LIN {X 0,Y 573.253,Z 369.075,A -85,B 0,C 180,E1 -2323.622,E2 -2323.622} C_VEL
LIN {X 0,Y 573.279,Z 369.074,A -85,B 0,C 180,E1 -2325.807,E2 -2325.807} C_VEL
LIN {X 0,Y 573.268,Z 369.074,A -85,B 0,C 180,E1 -2328.745,E2 -2328.745} C_VEL
LIN {X 0,Y 573.293,Z 369.076,A -85,B 0,C 180,E1 -2331.541,E2 -2331.541} C_VEL
LIN {X 0,Y 573.293,Z 369.073,A -85,B 0,C 180,E1 -2334.372,E2 -2334.372} C_VEL
LIN {X 0,Y 573.313,Z 369.07,A -85,B 0,C 180,E1 -2337.892,E2 -2337.892} C_VEL
LIN {X 0,Y 573.334,Z 369.065,A -85,B 0,C 180,E1 -2340.702,E2 -2340.702} C_VEL
LIN {X 0,Y 573.234,Z 369.083,A -85,B 0,C 180,E1 -2343.515,E2 -2343.515} C_VEL
LIN {X 0,Y 573.294,Z 369.071,A -85,B 0,C 180,E1 -2345.628,E2 -2345.628} C_VEL
LIN {X 0,Y 573.276,Z 369.072,A -85,B 0,C 180,E1 -2347.75,E2 -2347.75} C_VEL
LIN {X 0,Y 573.269,Z 369.075,A -85,B 0,C 180,E1 -2350.597,E2 -2350.597} C_VEL
LIN {X 0,Y 573.268,Z 369.073,A -85,B 0,C 180,E1 -2352.749,E2 -2352.749} C_VEL
LIN {X 0,Y 573.239,Z 369.079,A -85,B 0,C 180,E1 -2354.92,E2 -2354.92} C_VEL
LIN {X 0,Y 573.243,Z 369.077,A -85,B 0,C 180,E1 -2357.849,E2 -2357.849} C_VEL
LIN {X 0,Y 573.258,Z 369.077,A -85,B 0,C 180,E1 -2360.077,E2 -2360.077} C_VEL
LIN {X 0,Y 573.239,Z 369.076,A -85,B 0,C 180,E1 -2363.099,E2 -2363.099} C_VEL
LIN {X 0,Y 573.254,Z 369.076,A -85,B 0,C 180,E1 -2364.389,E2 -2364.389} C_VEL
LIN {X 0,Y 572.629,Z 369.154,A -85,B 0,C 180,E1 -2364.975,E2 -2364.975} C_VEL
LIN {X 0,Y 569.787,Z 369.513,A -85,B 0,C 180,E1 -2365.926,E2 -2365.926} C_VEL
LIN {X 0,Y 567.353,Z 369.819,A -85,B 0,C 180,E1 -2366.692,E2 -2366.692} C_VEL
LIN {X 0,Y 566.297,Z 369.948,A -85,B 0,C 180,E1 -2367.283,E2 -2367.283} C_VEL
LIN {X 0,Y 566.207,Z 369.957,A -85,B 0,C 180,E1 -2367.483,E2 -2367.483} C_VEL
LIN {X 0,Y 566.205,Z 369.954,A -85,B 0,C 180,E1 -2369.769,E2 -2369.769} C_VEL
LIN {X 0,Y 566.208,Z 369.959,A -85,B 0,C 180,E1 -2372.43,E2 -2372.43} C_VEL
LIN {X 0,Y 566.186,Z 369.955,A -85,B 0,C 180,E1 -2374.99,E2 -2374.99} C_VEL
LIN {X 0,Y 566.2,Z 369.959,A -85,B 0,C 180,E1 -2377.461,E2 -2377.461} C_VEL
LIN {X 0,Y 566.222,Z 369.951,A -85,B 0,C 180,E1 -2380.198,E2 -2380.198} C_VEL
LIN {X 0,Y 566.203,Z 369.957,A -85,B 0,C 180,E1 -2383.054,E2 -2383.054} C_VEL
LIN {X 0,Y 566.206,Z 369.96,A -85,B 0,C 180,E1 -2386.048,E2 -2386.048} C_VEL
LIN {X 0,Y 566.186,Z 369.955,A -85,B 0,C 180,E1 -2388.861,E2 -2388.861} C_VEL
LIN {X 0,Y 566.19,Z 369.958,A -85,B 0,C 180,E1 -2391.637,E2 -2391.637} C_VEL
LIN {X 0,Y 566.135,Z 369.965,A -85,B 0,C 180,E1 -2394.306,E2 -2394.306} C_VEL
LIN {X 0,Y 566.112,Z 369.972,A -85,B 0,C 180,E1 -2395.175,E2 -2395.175} C_VEL
LIN {X 0,Y 566.066,Z 370.716,A -85,B 0,C 180,E1 -2396.289,E2 -2396.289} C_VEL
LIN {X 0,Y 566.04,Z 373.544,A -85,B 0,C 180,E1 -2398.95,E2 -2398.95} C_VEL
LIN {X 0,Y 565.999,Z 376.682,A -85,B 0,C 180,E1 -2401.846,E2 -2401.846} C_VEL
LIN {X 0,Y 565.988,Z 379.352,A -85,B 0,C 180,E1 -2404.24,E2 -2404.24} C_VEL
LIN {X 0,Y 565.896,Z 382.829,A -85,B 0,C 180,E1 -2407.356,E2 -2407.356} C_VEL
LIN {X 0,Y 565.884,Z 385.612,A -85,B 0,C 180,E1 -2409.65,E2 -2409.65} C_VEL
LIN {X 0,Y 565.864,Z 389.455,A -85,B 0,C 180,E1 -2412.658,E2 -2412.658} C_VEL
LIN {X 0,Y 565.893,Z 393.314,A -85,B 0,C 180,E1 -2415.63,E2 -2415.63} C_VEL
LIN {X 0,Y 565.897,Z 395.671,A -85,B 0,C 180,E1 -2417.425,E2 -2417.425} C_VEL
LIN {X 0,Y 566.89,Z 403.279,A -85,B 0,C 180,E1 -2417.629,E2 -2417.629} C_VEL
LIN {X 0,Y 566.772,Z 415.78,A -85,B 0,C 180,E1 -2418.013,E2 -2418.013} C_VEL
LIN {X 0,Y 566.661,Z 428.299,A -85,B 0,C 180,E1 -2418.554,E2 -2418.554} C_VEL
LIN {X 0,Y 566.512,Z 439.58,A -85,B 0,C 180,E1 -2419.192,E2 -2419.192} C_VEL
LIN {X 0,Y 566.349,Z 450.842,A -85,B 0,C 180,E1 -2419.995,E2 -2419.995} C_VEL
LIN {X 0,Y 566.238,Z 460.89,A -85,B 0,C 180,E1 -2420.895,E2 -2420.895} C_VEL
LIN {X 0,Y 566.113,Z 470.591,A -85,B 0,C 180,E1 -2421.972,E2 -2421.972} C_VEL
LIN {X 0,Y 566.05,Z 477.159,A -85,B 0,C 180,E1 -2422.868,E2 -2422.868} C_VEL
LIN {X 0,Y 566.003,Z 483.628,A -85,B 0,C 180,E1 -2423.942,E2 -2423.942} C_VEL
LIN {X 0,Y 565.877,Z 488.765,A -85,B 0,C 180,E1 -2425.013,E2 -2425.013} C_VEL
LIN {X 0,Y 565.926,Z 492.754,A -85,B 0,C 180,E1 -2426.084,E2 -2426.084} C_VEL
LIN {X 0,Y 565.877,Z 495.702,A -85,B 0,C 180,E1 -2427.153,E2 -2427.153} C_VEL
LIN {X 0,Y 565.841,Z 497.128,A -85,B 0,C 180,E1 -2427.865,E2 -2427.865} C_VEL
LIN {X 0,Y 565.841,Z 498.756,A -85,B 0,C 180,E1 -2429.288,E2 -2429.288} C_VEL
LIN {X 0,Y 565.839,Z 498.996,A -85,B 0,C 180,E1 -2430,E2 -2430} C_VEL
LIN {X 0,Y 565.841,Z 498.814,A -85,B 0,C 180,E1 -2430.712,E2 -2430.712} C_VEL
LIN {X 0,Y 565.841,Z 497.268,A -85,B 0,C 180,E1 -2432.135,E2 -2432.135} C_VEL
LIN {X 0,Y 565.878,Z 495.907,A -85,B 0,C 180,E1 -2432.848,E2 -2432.848} C_VEL
LIN {X 0,Y 565.926,Z 493.03,A -85,B 0,C 180,E1 -2433.917,E2 -2433.917} C_VEL
LIN {X 0,Y 565.878,Z 489.129,A -85,B 0,C 180,E1 -2434.988,E2 -2434.988} C_VEL
LIN {X 0,Y 565.991,Z 484.096,A -85,B 0,C 180,E1 -2436.059,E2 -2436.059} C_VEL
LIN {X 0,Y 566.031,Z 477.771,A -85,B 0,C 180,E1 -2437.133,E2 -2437.133} C_VEL
LIN {X 0,Y 566.128,Z 469.849,A -85,B 0,C 180,E1 -2438.208,E2 -2438.208} C_VEL
LIN {X 0,Y 566.249,Z 459.997,A -85,B 0,C 180,E1 -2439.285,E2 -2439.285} C_VEL
LIN {X 0,Y 566.426,Z 449.677,A -85,B 0,C 180,E1 -2440.184,E2 -2440.184} C_VEL
LIN {X 0,Y 566.537,Z 438.407,A -85,B 0,C 180,E1 -2440.972,E2 -2440.972} C_VEL
LIN {X 0,Y 566.659,Z 427.185,A -85,B 0,C 180,E1 -2441.593,E2 -2441.593} C_VEL
LIN {X 0,Y 566.781,Z 414.589,A -85,B 0,C 180,E1 -2442.119,E2 -2442.119} C_VEL
LIN {X 0,Y 566.818,Z 401.411,A -85,B 0,C 180,E1 -2442.509,E2 -2442.509} C_VEL
LIN {X 0,Y 565.899,Z 395.669,A -85,B 0,C 180,E1 -2442.667,E2 -2442.667} C_VEL
LIN {X 0,Y 565.855,Z 392.455,A -85,B 0,C 180,E1 -2445.119,E2 -2445.119} C_VEL
LIN {X 0,Y 565.864,Z 389.571,A -85,B 0,C 180,E1 -2447.342,E2 -2447.342} C_VEL
LIN {X 0,Y 565.884,Z 385.726,A -85,B 0,C 180,E1 -2450.35,E2 -2450.35} C_VEL
LIN {X 0,Y 565.91,Z 382.308,A -85,B 0,C 180,E1 -2453.219,E2 -2453.219} C_VEL
LIN {X 0,Y 565.988,Z 379.451,A -85,B 0,C 180,E1 -2455.76,E2 -2455.76} C_VEL
LIN {X 0,Y 566.002,Z 376.782,A -85,B 0,C 180,E1 -2458.163,E2 -2458.163} C_VEL
LIN {X 0,Y 566.04,Z 373.651,A -85,B 0,C 180,E1 -2461.05,E2 -2461.05} C_VEL
LIN {X 0,Y 566.068,Z 370.535,A -85,B 0,C 180,E1 -2463.966,E2 -2463.966} C_VEL
LIN {X 0,Y 566.104,Z 369.973,A -85,B 0,C 180,E1 -2464.978,E2 -2464.978} C_VEL
LIN {X 0,Y 566.201,Z 369.957,A -85,B 0,C 180,E1 -2467.461,E2 -2467.461} C_VEL
LIN {X 0,Y 566.212,Z 369.955,A -85,B 0,C 180,E1 -2470.199,E2 -2470.199} C_VEL
LIN {X 0,Y 566.21,Z 369.953,A -85,B 0,C 180,E1 -2473.054,E2 -2473.054} C_VEL
LIN {X 0,Y 566.199,Z 369.957,A -85,B 0,C 180,E1 -2476.049,E2 -2476.049} C_VEL
LIN {X 0,Y 566.208,Z 369.959,A -85,B 0,C 180,E1 -2479.215,E2 -2479.215} C_VEL
LIN {X 0,Y 566.194,Z 369.955,A -85,B 0,C 180,E1 -2481.637,E2 -2481.637} C_VEL
LIN {X 0,Y 566.197,Z 369.96,A -85,B 0,C 180,E1 -2484.31,E2 -2484.31} C_VEL
LIN {X 0,Y 566.225,Z 369.951,A -85,B 0,C 180,E1 -2486.898,E2 -2486.898} C_VEL
LIN {X 0,Y 566.187,Z 369.962,A -85,B 0,C 180,E1 -2489.407,E2 -2489.407} C_VEL
LIN {X 0,Y 566.217,Z 369.952,A -85,B 0,C 180,E1 -2491.858,E2 -2491.858} C_VEL
LIN {X 0,Y 566.216,Z 369.957,A -85,B 0,C 180,E1 -2494.251,E2 -2494.251} C_VEL
LIN {X 0,Y 566.175,Z 369.957,A -85,B 0,C 180,E1 -2496.719,E2 -2496.719} C_VEL
LIN {X 0,Y 566.22,Z 369.958,A -85,B 0,C 180,E1 -2499.663,E2 -2499.663} C_VEL
LIN {X 0,Y 566.204,Z 369.957,A -85,B 0,C 180,E1 -2502.668,E2 -2502.668} C_VEL
LIN {X 0,Y 566.24,Z 369.949,A -85,B 0,C 180,E1 -2505.627,E2 -2505.627} C_VEL
LIN {X 0,Y 566.241,Z 369.949,A -85,B 0,C 180,E1 -2508.675,E2 -2508.675} C_VEL
LIN {X 0,Y 566.212,Z 369.957,A -85,B 0,C 180,E1 -2511.434,E2 -2511.434} C_VEL
LIN {X 0,Y 566.263,Z 369.947,A -85,B 0,C 180,E1 -2514.302,E2 -2514.302} C_VEL
LIN {X 0,Y 566.28,Z 369.945,A -85,B 0,C 180,E1 -2517.866,E2 -2517.866} C_VEL
LIN {X 0,Y 566.307,Z 369.941,A -85,B 0,C 180,E1 -2520.711,E2 -2520.711} C_VEL
LIN {X 0,Y 566.276,Z 369.944,A -85,B 0,C 180,E1 -2522.846,E2 -2522.846} C_VEL
LIN {X 0,Y 566.262,Z 369.948,A -85,B 0,C 180,E1 -2525.698,E2 -2525.698} C_VEL
LIN {X 0,Y 566.238,Z 369.955,A -85,B 0,C 180,E1 -2528.566,E2 -2528.566} C_VEL
LIN {X 0,Y 566.248,Z 369.949,A -85,B 0,C 180,E1 -2531.454,E2 -2531.454} C_VEL
LIN {X 0,Y 566.241,Z 369.949,A -85,B 0,C 180,E1 -2534.507,E2 -2534.507} C_VEL
LIN {X 0,Y 566.203,Z 369.959,A -85,B 0,C 180,E1 -2537.332,E2 -2537.332} C_VEL
LIN {X 0,Y 566.219,Z 369.955,A -85,B 0,C 180,E1 -2540.337,E2 -2540.337} C_VEL
LIN {X 0,Y 566.174,Z 369.958,A -85,B 0,C 180,E1 -2543.281,E2 -2543.281} C_VEL
LIN {X 0,Y 566.219,Z 369.958,A -85,B 0,C 180,E1 -2545.749,E2 -2545.749} C_VEL
LIN {X 0,Y 566.208,Z 369.953,A -85,B 0,C 180,E1 -2548.202,E2 -2548.202} C_VEL
LIN {X 0,Y 566.196,Z 369.959,A -85,B 0,C 180,E1 -2551.076,E2 -2551.076} C_VEL
LIN {X 0,Y 566.217,Z 369.953,A -85,B 0,C 180,E1 -2553.734,E2 -2553.734} C_VEL
LIN {X 0,Y 566.204,Z 369.955,A -85,B 0,C 180,E1 -2556.57,E2 -2556.57} C_VEL
LIN {X 0,Y 566.226,Z 369.955,A -85,B 0,C 180,E1 -2559.686,E2 -2559.686} C_VEL
LIN {X 0,Y 566.206,Z 369.96,A -85,B 0,C 180,E1 -2562.917,E2 -2562.917} C_VEL
LIN {X 0,Y 566.207,Z 369.957,A -85,B 0,C 180,E1 -2566.048,E2 -2566.048} C_VEL
LIN {X 0,Y 566.186,Z 369.956,A -85,B 0,C 180,E1 -2568.861,E2 -2568.861} C_VEL
LIN {X 0,Y 566.189,Z 369.962,A -85,B 0,C 180,E1 -2571.637,E2 -2571.637} C_VEL
LIN {X 0,Y 566.243,Z 370.1,A -85,B 0,C 180,E1 -2573.045,E2 -2573.045} C_VEL
LIN {X 0,Y 566.803,Z 373.915,A -85,B 0,C 180,E1 -2574.354,E2 -2574.354} C_VEL
LIN {X 0,Y 566.814,Z 381.859,A -85,B 0,C 180,E1 -2576.937,E2 -2576.937} C_VEL
LIN {X 0,Y 566.649,Z 391.126,A -85,B 0,C 180,E1 -2579.847,E2 -2579.847} C_VEL
LIN {X 0,Y 566.525,Z 400.394,A -85,B 0,C 180,E1 -2582.677,E2 -2582.677} C_VEL
LIN {X 0,Y 566.399,Z 410.985,A -85,B 0,C 180,E1 -2585.828,E2 -2585.828} C_VEL
LIN {X 0,Y 566.252,Z 420.416,A -85,B 0,C 180,E1 -2588.569,E2 -2588.569} C_VEL
LIN {X 0,Y 566.186,Z 429.52,A -85,B 0,C 180,E1 -2591.171,E2 -2591.171} C_VEL
LIN {X 0,Y 566.116,Z 440.111,A -85,B 0,C 180,E1 -2594.15,E2 -2594.15} C_VEL
LIN {X 0,Y 566.028,Z 450.702,A -85,B 0,C 180,E1 -2597.085,E2 -2597.085} C_VEL
LIN {X 0,Y 566.04,Z 451.53,A -85,B 0,C 180,E1 -2597.314,E2 -2597.314} C_VEL
LIN {X 0,Y 566.944,Z 458.363,A -85,B 0,C 180,E1 -2597.471,E2 -2597.471} C_VEL
LIN {X 0,Y 566.832,Z 470.492,A -85,B 0,C 180,E1 -2597.786,E2 -2597.786} C_VEL
LIN {X 0,Y 566.746,Z 482.316,A -85,B 0,C 180,E1 -2598.229,E2 -2598.229} C_VEL
LIN {X 0,Y 566.59,Z 493.421,A -85,B 0,C 180,E1 -2598.779,E2 -2598.779} C_VEL
LIN {X 0,Y 566.423,Z 505.476,A -85,B 0,C 180,E1 -2599.545,E2 -2599.545} C_VEL
LIN {X 0,Y 566.301,Z 515.645,A -85,B 0,C 180,E1 -2600.355,E2 -2600.355} C_VEL
LIN {X 0,Y 566.166,Z 524.786,A -85,B 0,C 180,E1 -2601.253,E2 -2601.253} C_VEL
LIN {X 0,Y 566.081,Z 533.689,A -85,B 0,C 180,E1 -2602.33,E2 -2602.33} C_VEL
LIN {X 0,Y 565.968,Z 540.955,A -85,B 0,C 180,E1 -2603.422,E2 -2603.422} C_VEL
LIN {X 0,Y 566.004,Z 545.68,A -85,B 0,C 180,E1 -2604.299,E2 -2604.299} C_VEL
LIN {X 0,Y 565.933,Z 550.371,A -85,B 0,C 180,E1 -2605.37,E2 -2605.37} C_VEL
LIN {X 0,Y 565.927,Z 553.956,A -85,B 0,C 180,E1 -2606.44,E2 -2606.44} C_VEL
LIN {X 0,Y 565.878,Z 555.808,A -85,B 0,C 180,E1 -2607.152,E2 -2607.152} C_VEL
LIN {X 0,Y 565.84,Z 557.2,A -85,B 0,C 180,E1 -2607.864,E2 -2607.864} C_VEL
LIN {X 0,Y 565.841,Z 558.784,A -85,B 0,C 180,E1 -2609.288,E2 -2609.288} C_VEL
LIN {X 0,Y 565.839,Z 559,A -85,B 0,C 180,E1 -2610,E2 -2610} C_VEL
LIN {X 0,Y 565.846,Z 558.185,A -85,B 0,C 180,E1 -2611.423,E2 -2611.423} C_VEL
LIN {X 0,Y 565.84,Z 557.201,A -85,B 0,C 180,E1 -2612.135,E2 -2612.135} C_VEL
LIN {X 0,Y 565.878,Z 555.81,A -85,B 0,C 180,E1 -2612.847,E2 -2612.847} C_VEL
LIN {X 0,Y 565.926,Z 552.896,A -85,B 0,C 180,E1 -2613.916,E2 -2613.916} C_VEL
LIN {X 0,Y 565.878,Z 548.95,A -85,B 0,C 180,E1 -2614.987,E2 -2614.987} C_VEL
LIN {X 0,Y 566.002,Z 543.867,A -85,B 0,C 180,E1 -2616.058,E2 -2616.058} C_VEL
LIN {X 0,Y 566.04,Z 537.47,A -85,B 0,C 180,E1 -2617.132,E2 -2617.132} C_VEL
LIN {X 0,Y 566.134,Z 529.478,A -85,B 0,C 180,E1 -2618.208,E2 -2618.208} C_VEL
LIN {X 0,Y 566.229,Z 521.337,A -85,B 0,C 180,E1 -2619.105,E2 -2619.105} C_VEL
LIN {X 0,Y 566.35,Z 511.402,A -85,B 0,C 180,E1 -2620.005,E2 -2620.005} C_VEL
LIN {X 0,Y 566.523,Z 500.286,A -85,B 0,C 180,E1 -2620.807,E2 -2620.807} C_VEL
LIN {X 0,Y 566.613,Z 489.178,A -85,B 0,C 180,E1 -2621.447,E2 -2621.447} C_VEL
LIN {X 0,Y 566.748,Z 476.989,A -85,B 0,C 180,E1 -2621.988,E2 -2621.988} C_VEL
LIN {X 0,Y 566.893,Z 464.178,A -85,B 0,C 180,E1 -2622.394,E2 -2622.394} C_VEL
LIN {X 0,Y 566.752,Z 456.087,A -85,B 0,C 180,E1 -2622.579,E2 -2622.579} C_VEL
LIN {X 0,Y 566.04,Z 451.53,A -85,B 0,C 180,E1 -2622.686,E2 -2622.686} C_VEL
LIN {X 0,Y 566.093,Z 441.435,A -85,B 0,C 180,E1 -2625.481,E2 -2625.481} C_VEL
LIN {X 0,Y 566.167,Z 430.844,A -85,B 0,C 180,E1 -2628.454,E2 -2628.454} C_VEL
LIN {X 0,Y 566.245,Z 421.577,A -85,B 0,C 180,E1 -2631.096,E2 -2631.096} C_VEL
LIN {X 0,Y 566.363,Z 412.309,A -85,B 0,C 180,E1 -2633.784,E2 -2633.784} C_VEL
LIN {X 0,Y 566.496,Z 403.042,A -85,B 0,C 180,E1 -2636.527,E2 -2636.527} C_VEL
LIN {X 0,Y 566.571,Z 393.775,A -85,B 0,C 180,E1 -2639.339,E2 -2639.339} C_VEL
LIN {X 0,Y 566.777,Z 384.507,A -85,B 0,C 180,E1 -2642.222,E2 -2642.222} C_VEL
LIN {X 0,Y 566.848,Z 376.564,A -85,B 0,C 180,E1 -2644.773,E2 -2644.773} C_VEL
LIN {X 0,Y 566.593,Z 372.083,A -85,B 0,C 180,E1 -2646.268,E2 -2646.268} C_VEL
LIN {X 0,Y 566.237,Z 369.956,A -85,B 0,C 180,E1 -2647.011,E2 -2647.011} C_VEL
LIN {X 0,Y 566.217,Z 369.954,A -85,B 0,C 180,E1 -2649.686,E2 -2649.686} C_VEL
LIN {X 0,Y 566.218,Z 369.96,A -85,B 0,C 180,E1 -2652.087,E2 -2652.087} C_VEL
LIN {X 0,Y 566.176,Z 369.961,A -85,B 0,C 180,E1 -2655.036,E2 -2655.036} C_VEL
LIN {X 0,Y 566.192,Z 369.954,A -85,B 0,C 180,E1 -2657.911,E2 -2657.911} C_VEL
LIN {X 0,Y 566.225,Z 369.956,A -85,B 0,C 180,E1 -2660.727,E2 -2660.727} C_VEL
LIN {X 0,Y 566.205,Z 369.958,A -85,B 0,C 180,E1 -2663.786,E2 -2663.786} C_VEL
LIN {X 0,Y 566.215,Z 369.953,A -85,B 0,C 180,E1 -2666.266,E2 -2666.266} C_VEL
LIN {X 0,Y 566.195,Z 369.959,A -85,B 0,C 180,E1 -2668.924,E2 -2668.924} C_VEL
LIN {X 0,Y 566.216,Z 369.952,A -85,B 0,C 180,E1 -2671.857,E2 -2671.857} C_VEL
LIN {X 0,Y 566.218,Z 369.958,A -85,B 0,C 180,E1 -2674.251,E2 -2674.251} C_VEL
LIN {X 0,Y 566.173,Z 369.958,A -85,B 0,C 180,E1 -2676.719,E2 -2676.719} C_VEL
LIN {X 0,Y 566.218,Z 369.956,A -85,B 0,C 180,E1 -2679.663,E2 -2679.663} C_VEL
LIN {X 0,Y 566.203,Z 369.959,A -85,B 0,C 180,E1 -2682.668,E2 -2682.668} C_VEL
LIN {X 0,Y 566.239,Z 369.949,A -85,B 0,C 180,E1 -2685.627,E2 -2685.627} C_VEL
LIN {X 0,Y 566.239,Z 369.95,A -85,B 0,C 180,E1 -2688.675,E2 -2688.675} C_VEL
LIN {X 0,Y 566.237,Z 369.955,A -85,B 0,C 180,E1 -2691.434,E2 -2691.434} C_VEL
LIN {X 0,Y 566.261,Z 369.948,A -85,B 0,C 180,E1 -2694.302,E2 -2694.302} C_VEL
LIN {X 0,Y 566.285,Z 369.945,A -85,B 0,C 180,E1 -2697.866,E2 -2697.866} C_VEL
LIN {X 0,Y 566.305,Z 369.941,A -85,B 0,C 180,E1 -2700.711,E2 -2700.711} C_VEL
LIN {X 0,Y 566.275,Z 369.946,A -85,B 0,C 180,E1 -2702.846,E2 -2702.846} C_VEL
LIN {X 0,Y 566.262,Z 369.947,A -85,B 0,C 180,E1 -2705.698,E2 -2705.698} C_VEL
LIN {X 0,Y 566.212,Z 369.958,A -85,B 0,C 180,E1 -2708.566,E2 -2708.566} C_VEL
LIN {X 0,Y 566.247,Z 369.949,A -85,B 0,C 180,E1 -2711.454,E2 -2711.454} C_VEL
LIN {X 0,Y 566.239,Z 369.949,A -85,B 0,C 180,E1 -2714.506,E2 -2714.506} C_VEL
LIN {X 0,Y 566.202,Z 369.958,A -85,B 0,C 180,E1 -2717.332,E2 -2717.332} C_VEL
LIN {X 0,Y 566.219,Z 369.957,A -85,B 0,C 180,E1 -2720.337,E2 -2720.337} C_VEL
LIN {X 0,Y 566.174,Z 369.957,A -85,B 0,C 180,E1 -2723.281,E2 -2723.281} C_VEL
LIN {X 0,Y 566.218,Z 369.957,A -85,B 0,C 180,E1 -2725.749,E2 -2725.749} C_VEL
LIN {X 0,Y 566.207,Z 369.957,A -85,B 0,C 180,E1 -2727.483,E2 -2727.483} C_VEL
LIN {X 0,Y 565.527,Z 370.039,A -85,B 0,C 180,E1 -2728.077,E2 -2728.077} C_VEL
LIN {X 0,Y 562.661,Z 370.401,A -85,B 0,C 180,E1 -2729.041,E2 -2729.041} C_VEL
LIN {X 0,Y 560.252,Z 370.698,A -85,B 0,C 180,E1 -2729.816,E2 -2729.816} C_VEL
LIN {X 0,Y 559.224,Z 370.827,A -85,B 0,C 180,E1 -2730.415,E2 -2730.415} C_VEL
LIN {X 0,Y 559.144,Z 370.834,A -85,B 0,C 180,E1 -2730.618,E2 -2730.618} C_VEL
LIN {X 0,Y 559.167,Z 370.831,A -85,B 0,C 180,E1 -2733.575,E2 -2733.575} C_VEL
LIN {X 0,Y 559.151,Z 370.832,A -85,B 0,C 180,E1 -2736.445,E2 -2736.445} C_VEL
LIN {X 0,Y 559.182,Z 370.831,A -85,B 0,C 180,E1 -2738.934,E2 -2738.934} C_VEL
LIN {X 0,Y 559.169,Z 370.831,A -85,B 0,C 180,E1 -2741.77,E2 -2741.77} C_VEL
LIN {X 0,Y 559.139,Z 370.837,A -85,B 0,C 180,E1 -2744.74,E2 -2744.74} C_VEL
LIN {X 0,Y 559.168,Z 370.831,A -85,B 0,C 180,E1 -2747.257,E2 -2747.257} C_VEL
LIN {X 0,Y 559.183,Z 370.829,A -85,B 0,C 180,E1 -2750.134,E2 -2750.134} C_VEL
LIN {X 0,Y 559.142,Z 370.838,A -85,B 0,C 180,E1 -2752.891,E2 -2752.891} C_VEL
LIN {X 0,Y 559.006,Z 370.857,A -85,B 0,C 180,E1 -2755.545,E2 -2755.545} C_VEL
LIN {X 0,Y 558.982,Z 372.599,A -85,B 0,C 180,E1 -2757.393,E2 -2757.393} C_VEL
LIN {X 0,Y 558.969,Z 375.521,A -85,B 0,C 180,E1 -2760.175,E2 -2760.175} C_VEL
LIN {X 0,Y 558.917,Z 378.691,A -85,B 0,C 180,E1 -2763.084,E2 -2763.084} C_VEL
LIN {X 0,Y 558.856,Z 381.355,A -85,B 0,C 180,E1 -2765.481,E2 -2765.481} C_VEL
LIN {X 0,Y 558.837,Z 384.778,A -85,B 0,C 180,E1 -2768.534,E2 -2768.534} C_VEL
LIN {X 0,Y 558.789,Z 387.534,A -85,B 0,C 180,E1 -2770.913,E2 -2770.913} C_VEL
LIN {X 0,Y 558.771,Z 391.378,A -85,B 0,C 180,E1 -2773.936,E2 -2773.936} C_VEL
LIN {X 0,Y 558.784,Z 394.26,A -85,B 0,C 180,E1 -2776.174,E2 -2776.174} C_VEL
LIN {X 0,Y 558.804,Z 395.672,A -85,B 0,C 180,E1 -2777.262,E2 -2777.262} C_VEL
LIN {X 0,Y 559.966,Z 404.216,A -85,B 0,C 180,E1 -2777.496,E2 -2777.496} C_VEL
LIN {X 0,Y 559.838,Z 416.298,A -85,B 0,C 180,E1 -2777.88,E2 -2777.88} C_VEL
LIN {X 0,Y 559.688,Z 428.309,A -85,B 0,C 180,E1 -2778.41,E2 -2778.41} C_VEL
LIN {X 0,Y 559.516,Z 439.666,A -85,B 0,C 180,E1 -2779.06,E2 -2779.06} C_VEL
LIN {X 0,Y 559.353,Z 450.85,A -85,B 0,C 180,E1 -2779.869,E2 -2779.869} C_VEL
LIN {X 0,Y 559.211,Z 460.895,A -85,B 0,C 180,E1 -2780.779,E2 -2780.779} C_VEL
LIN {X 0,Y 559.05,Z 470.595,A -85,B 0,C 180,E1 -2781.87,E2 -2781.87} C_VEL
LIN {X 0,Y 558.971,Z 478.456,A -85,B 0,C 180,E1 -2782.977,E2 -2782.977} C_VEL
LIN {X 0,Y 558.936,Z 485.455,A -85,B 0,C 180,E1 -2784.227,E2 -2784.227} C_VEL
LIN {X 0,Y 558.826,Z 490.195,A -85,B 0,C 180,E1 -2785.311,E2 -2785.311} C_VEL
LIN {X 0,Y 558.836,Z 493.828,A -85,B 0,C 180,E1 -2786.395,E2 -2786.395} C_VEL
LIN {X 0,Y 558.799,Z 495.704,A -85,B 0,C 180,E1 -2787.116,E2 -2787.116} C_VEL
LIN {X 0,Y 558.747,Z 497.128,A -85,B 0,C 180,E1 -2787.838,E2 -2787.838} C_VEL
LIN {X 0,Y 558.741,Z 498.757,A -85,B 0,C 180,E1 -2789.279,E2 -2789.279} C_VEL
LIN {X 0,Y 558.74,Z 498.996,A -85,B 0,C 180,E1 -2790,E2 -2790} C_VEL
LIN {X 0,Y 558.741,Z 498.814,A -85,B 0,C 180,E1 -2790.721,E2 -2790.721} C_VEL
LIN {X 0,Y 558.747,Z 497.267,A -85,B 0,C 180,E1 -2792.163,E2 -2792.163} C_VEL
LIN {X 0,Y 558.8,Z 495.905,A -85,B 0,C 180,E1 -2792.884,E2 -2792.884} C_VEL
LIN {X 0,Y 558.844,Z 493.028,A -85,B 0,C 180,E1 -2793.966,E2 -2793.966} C_VEL
LIN {X 0,Y 558.798,Z 489.126,A -85,B 0,C 180,E1 -2795.051,E2 -2795.051} C_VEL
LIN {X 0,Y 558.91,Z 484.093,A -85,B 0,C 180,E1 -2796.136,E2 -2796.136} C_VEL
LIN {X 0,Y 558.973,Z 477.767,A -85,B 0,C 180,E1 -2797.223,E2 -2797.223} C_VEL
LIN {X 0,Y 559.091,Z 469.844,A -85,B 0,C 180,E1 -2798.312,E2 -2798.312} C_VEL
LIN {X 0,Y 559.224,Z 459.991,A -85,B 0,C 180,E1 -2799.403,E2 -2799.403} C_VEL
LIN {X 0,Y 559.424,Z 449.671,A -85,B 0,C 180,E1 -2800.313,E2 -2800.313} C_VEL
LIN {X 0,Y 559.546,Z 438.706,A -85,B 0,C 180,E1 -2801.091,E2 -2801.091} C_VEL
LIN {X 0,Y 559.684,Z 428.451,A -85,B 0,C 180,E1 -2801.673,E2 -2801.673} C_VEL
LIN {X 0,Y 559.824,Z 415.741,A -85,B 0,C 180,E1 -2802.231,E2 -2802.231} C_VEL
LIN {X 0,Y 559.879,Z 402.303,A -85,B 0,C 180,E1 -2802.644,E2 -2802.644} C_VEL
LIN {X 0,Y 558.786,Z 395.669,A -85,B 0,C 180,E1 -2802.831,E2 -2802.831} C_VEL
LIN {X 0,Y 558.753,Z 392.454,A -85,B 0,C 180,E1 -2805.316,E2 -2805.316} C_VEL
LIN {X 0,Y 558.775,Z 389.57,A -85,B 0,C 180,E1 -2807.57,E2 -2807.57} C_VEL
LIN {X 0,Y 558.793,Z 386.687,A -85,B 0,C 180,E1 -2809.852,E2 -2809.852} C_VEL
LIN {X 0,Y 558.808,Z 384.072,A -85,B 0,C 180,E1 -2812.167,E2 -2812.167} C_VEL
LIN {X 0,Y 558.888,Z 380.77,A -85,B 0,C 180,E1 -2815.123,E2 -2815.123} C_VEL
LIN {X 0,Y 558.906,Z 377.902,A -85,B 0,C 180,E1 -2817.727,E2 -2817.727} C_VEL
LIN {X 0,Y 558.964,Z 375.24,A -85,B 0,C 180,E1 -2820.194,E2 -2820.194} C_VEL
LIN {X 0,Y 558.98,Z 372.574,A -85,B 0,C 180,E1 -2822.727,E2 -2822.727} C_VEL
LIN {X 0,Y 559.006,Z 370.857,A -85,B 0,C 180,E1 -2824.455,E2 -2824.455} C_VEL
LIN {X 0,Y 559.143,Z 370.839,A -85,B 0,C 180,E1 -2827.109,E2 -2827.109} C_VEL
LIN {X 0,Y 559.165,Z 370.831,A -85,B 0,C 180,E1 -2829.942,E2 -2829.942} C_VEL
LIN {X 0,Y 559.169,Z 370.831,A -85,B 0,C 180,E1 -2832.743,E2 -2832.743} C_VEL
LIN {X 0,Y 559.153,Z 370.838,A -85,B 0,C 180,E1 -2835.761,E2 -2835.761} C_VEL
LIN {X 0,Y 559.167,Z 370.831,A -85,B 0,C 180,E1 -2838.23,E2 -2838.23} C_VEL
LIN {X 0,Y 559.183,Z 370.83,A -85,B 0,C 180,E1 -2841.191,E2 -2841.191} C_VEL
LIN {X 0,Y 559.161,Z 370.832,A -85,B 0,C 180,E1 -2843.791,E2 -2843.791} C_VEL
LIN {X 0,Y 559.168,Z 370.831,A -85,B 0,C 180,E1 -2846.425,E2 -2846.425} C_VEL
LIN {X 0,Y 559.161,Z 370.834,A -85,B 0,C 180,E1 -2848.981,E2 -2848.981} C_VEL
LIN {X 0,Y 559.174,Z 370.831,A -85,B 0,C 180,E1 -2851.619,E2 -2851.619} C_VEL
LIN {X 0,Y 559.184,Z 370.829,A -85,B 0,C 180,E1 -2853.903,E2 -2853.903} C_VEL
LIN {X 0,Y 559.145,Z 370.834,A -85,B 0,C 180,E1 -2856.572,E2 -2856.572} C_VEL
LIN {X 0,Y 559.186,Z 370.832,A -85,B 0,C 180,E1 -2859.396,E2 -2859.396} C_VEL
LIN {X 0,Y 559.148,Z 370.835,A -85,B 0,C 180,E1 -2861.686,E2 -2861.686} C_VEL
LIN {X 0,Y 559.167,Z 370.831,A -85,B 0,C 180,E1 -2863.948,E2 -2863.948} C_VEL
LIN {X 0,Y 559.177,Z 370.833,A -85,B 0,C 180,E1 -2866.184,E2 -2866.184} C_VEL
LIN {X 0,Y 559.199,Z 370.826,A -85,B 0,C 180,E1 -2869.134,E2 -2869.134} C_VEL
LIN {X 0,Y 559.201,Z 370.827,A -85,B 0,C 180,E1 -2872.053,E2 -2872.053} C_VEL
LIN {X 0,Y 559.258,Z 370.824,A -85,B 0,C 180,E1 -2874.953,E2 -2874.953} C_VEL
LIN {X 0,Y 559.252,Z 370.821,A -85,B 0,C 180,E1 -2877.839,E2 -2877.839} C_VEL
LIN {X 0,Y 559.277,Z 370.817,A -85,B 0,C 180,E1 -2880.72,E2 -2880.72} C_VEL
LIN {X 0,Y 559.243,Z 370.82,A -85,B 0,C 180,E1 -2882.881,E2 -2882.881} C_VEL
LIN {X 0,Y 559.232,Z 370.823,A -85,B 0,C 180,E1 -2885.77,E2 -2885.77} C_VEL
LIN {X 0,Y 559.196,Z 370.832,A -85,B 0,C 180,E1 -2888.674,E2 -2888.674} C_VEL
LIN {X 0,Y 559.211,Z 370.826,A -85,B 0,C 180,E1 -2891.6,E2 -2891.6} C_VEL
LIN {X 0,Y 559.206,Z 370.825,A -85,B 0,C 180,E1 -2894.595,E2 -2894.595} C_VEL
LIN {X 0,Y 559.146,Z 370.835,A -85,B 0,C 180,E1 -2897.557,E2 -2897.557} C_VEL
LIN {X 0,Y 559.178,Z 370.829,A -85,B 0,C 180,E1 -2899.837,E2 -2899.837} C_VEL
LIN {X 0,Y 559.146,Z 370.838,A -85,B 0,C 180,E1 -2902.153,E2 -2902.153} C_VEL
LIN {X 0,Y 559.181,Z 370.83,A -85,B 0,C 180,E1 -2905.298,E2 -2905.298} C_VEL
LIN {X 0,Y 559.186,Z 370.831,A -85,B 0,C 180,E1 -2907.712,E2 -2907.712} C_VEL
LIN {X 0,Y 559.158,Z 370.831,A -85,B 0,C 180,E1 -2910.183,E2 -2910.183} C_VEL
LIN {X 0,Y 559.162,Z 370.837,A -85,B 0,C 180,E1 -2912.715,E2 -2912.715} C_VEL
LIN {X 0,Y 559.133,Z 370.835,A -85,B 0,C 180,E1 -2915.324,E2 -2915.324} C_VEL
LIN {X 0,Y 559.139,Z 370.837,A -85,B 0,C 180,E1 -2918.017,E2 -2918.017} C_VEL
LIN {X 0,Y 559.16,Z 370.833,A -85,B 0,C 180,E1 -2920.812,E2 -2920.812} C_VEL
LIN {X 0,Y 559.145,Z 370.833,A -85,B 0,C 180,E1 -2923.734,E2 -2923.734} C_VEL
LIN {X 0,Y 559.173,Z 370.832,A -85,B 0,C 180,E1 -2926.801,E2 -2926.801} C_VEL
LIN {X 0,Y 559.163,Z 370.833,A -85,B 0,C 180,E1 -2929.188,E2 -2929.188} C_VEL
LIN {X 0,Y 559.136,Z 370.839,A -85,B 0,C 180,E1 -2931.982,E2 -2931.982} C_VEL
LIN {X 0,Y 559.204,Z 370.948,A -85,B 0,C 180,E1 -2932.798,E2 -2932.798} C_VEL
LIN {X 0,Y 559.852,Z 375.234,A -85,B 0,C 180,E1 -2934.287,E2 -2934.287} C_VEL
LIN {X 0,Y 559.864,Z 381.859,A -85,B 0,C 180,E1 -2936.472,E2 -2936.472} C_VEL
LIN {X 0,Y 559.685,Z 389.802,A -85,B 0,C 180,E1 -2939.013,E2 -2939.013} C_VEL
LIN {X 0,Y 559.564,Z 399.153,A -85,B 0,C 180,E1 -2941.927,E2 -2941.927} C_VEL
LIN {X 0,Y 559.408,Z 408.507,A -85,B 0,C 180,E1 -2944.764,E2 -2944.764} C_VEL
LIN {X 0,Y 559.289,Z 417.604,A -85,B 0,C 180,E1 -2947.464,E2 -2947.464} C_VEL
LIN {X 0,Y 559.18,Z 428.035,A -85,B 0,C 180,E1 -2950.499,E2 -2950.499} C_VEL
LIN {X 0,Y 559.059,Z 438.787,A -85,B 0,C 180,E1 -2953.569,E2 -2953.569} C_VEL
LIN {X 0,Y 558.997,Z 448.054,A -85,B 0,C 180,E1 -2956.18,E2 -2956.18} C_VEL
LIN {X 0,Y 558.962,Z 451.53,A -85,B 0,C 180,E1 -2957.15,E2 -2957.15} C_VEL
LIN {X 0,Y 560.019,Z 459.502,A -85,B 0,C 180,E1 -2957.336,E2 -2957.336} C_VEL
LIN {X 0,Y 559.902,Z 471.873,A -85,B 0,C 180,E1 -2957.679,E2 -2957.679} C_VEL
LIN {X 0,Y 559.772,Z 484.279,A -85,B 0,C 180,E1 -2958.172,E2 -2958.172} C_VEL
LIN {X 0,Y 559.63,Z 495.348,A -85,B 0,C 180,E1 -2958.75,E2 -2958.75} C_VEL
LIN {X 0,Y 559.427,Z 506.745,A -85,B 0,C 180,E1 -2959.504,E2 -2959.504} C_VEL
LIN {X 0,Y 559.244,Z 517.599,A -85,B 0,C 180,E1 -2960.415,E2 -2960.415} C_VEL
LIN {X 0,Y 559.127,Z 526.412,A -85,B 0,C 180,E1 -2961.325,E2 -2961.325} C_VEL
LIN {X 0,Y 558.996,Z 534.999,A -85,B 0,C 180,E1 -2962.414,E2 -2962.414} C_VEL
LIN {X 0,Y 558.885,Z 542.688,A -85,B 0,C 180,E1 -2963.649,E2 -2963.649} C_VEL
LIN {X 0,Y 558.869,Z 547.365,A -85,B 0,C 180,E1 -2964.588,E2 -2964.588} C_VEL
LIN {X 0,Y 558.868,Z 551.677,A -85,B 0,C 180,E1 -2965.673,E2 -2965.673} C_VEL
LIN {X 0,Y 558.836,Z 553.956,A -85,B 0,C 180,E1 -2966.395,E2 -2966.395} C_VEL
LIN {X 0,Y 558.799,Z 555.808,A -85,B 0,C 180,E1 -2967.116,E2 -2967.116} C_VEL
LIN {X 0,Y 558.746,Z 557.199,A -85,B 0,C 180,E1 -2967.837,E2 -2967.837} C_VEL
LIN {X 0,Y 558.741,Z 558.784,A -85,B 0,C 180,E1 -2969.279,E2 -2969.279} C_VEL
LIN {X 0,Y 558.74,Z 559,A -85,B 0,C 180,E1 -2970,E2 -2970} C_VEL
LIN {X 0,Y 558.746,Z 558.186,A -85,B 0,C 180,E1 -2971.441,E2 -2971.441} C_VEL
LIN {X 0,Y 558.746,Z 557.201,A -85,B 0,C 180,E1 -2972.162,E2 -2972.162} C_VEL
LIN {X 0,Y 558.799,Z 555.81,A -85,B 0,C 180,E1 -2972.884,E2 -2972.884} C_VEL
LIN {X 0,Y 558.843,Z 552.896,A -85,B 0,C 180,E1 -2973.966,E2 -2973.966} C_VEL
LIN {X 0,Y 558.798,Z 548.949,A -85,B 0,C 180,E1 -2975.051,E2 -2975.051} C_VEL
LIN {X 0,Y 558.921,Z 543.867,A -85,B 0,C 180,E1 -2976.136,E2 -2976.136} C_VEL
LIN {X 0,Y 558.977,Z 537.469,A -85,B 0,C 180,E1 -2977.223,E2 -2977.223} C_VEL
LIN {X 0,Y 559.099,Z 529.478,A -85,B 0,C 180,E1 -2978.312,E2 -2978.312} C_VEL
LIN {X 0,Y 559.195,Z 521.337,A -85,B 0,C 180,E1 -2979.221,E2 -2979.221} C_VEL
LIN {X 0,Y 559.359,Z 511.402,A -85,B 0,C 180,E1 -2980.131,E2 -2980.131} C_VEL
LIN {X 0,Y 559.527,Z 500.393,A -85,B 0,C 180,E1 -2980.937,E2 -2980.937} C_VEL
LIN {X 0,Y 559.672,Z 488.466,A -85,B 0,C 180,E1 -2981.628,E2 -2981.628} C_VEL
LIN {X 0,Y 559.825,Z 475.767,A -85,B 0,C 180,E1 -2982.185,E2 -2982.185} C_VEL
LIN {X 0,Y 559.959,Z 462.349,A -85,B 0,C 180,E1 -2982.596,E2 -2982.596} C_VEL
LIN {X 0,Y 559.833,Z 456.944,A -85,B 0,C 180,E1 -2982.72,E2 -2982.72} C_VEL
LIN {X 0,Y 558.962,Z 451.53,A -85,B 0,C 180,E1 -2982.849,E2 -2982.849} C_VEL
LIN {X 0,Y 559.056,Z 441.435,A -85,B 0,C 180,E1 -2985.681,E2 -2985.681} C_VEL
LIN {X 0,Y 559.134,Z 430.844,A -85,B 0,C 180,E1 -2988.694,E2 -2988.694} C_VEL
LIN {X 0,Y 559.227,Z 420.916,A -85,B 0,C 180,E1 -2991.567,E2 -2991.567} C_VEL
LIN {X 0,Y 559.396,Z 410.985,A -85,B 0,C 180,E1 -2994.494,E2 -2994.494} C_VEL
LIN {X 0,Y 559.521,Z 401.719,A -85,B 0,C 180,E1 -2997.288,E2 -2997.288} C_VEL
LIN {X 0,Y 559.657,Z 392.451,A -85,B 0,C 180,E1 -3000.153,E2 -3000.153} C_VEL
LIN {X 0,Y 559.848,Z 383.185,A -85,B 0,C 180,E1 -3003.098,E2 -3003.098} C_VEL
LIN {X 0,Y 559.896,Z 376.397,A -85,B 0,C 180,E1 -3005.323,E2 -3005.323} C_VEL
LIN {X 0,Y 559.263,Z 371.238,A -85,B 0,C 180,E1 -3007.099,E2 -3007.099} C_VEL
LIN {X 0,Y 559.174,Z 370.835,A -85,B 0,C 180,E1 -3007.302,E2 -3007.302} C_VEL
LIN {X 0,Y 559.163,Z 370.835,A -85,B 0,C 180,E1 -3009.942,E2 -3009.942} C_VEL
LIN {X 0,Y 559.168,Z 370.832,A -85,B 0,C 180,E1 -3012.743,E2 -3012.743} C_VEL
LIN {X 0,Y 559.153,Z 370.834,A -85,B 0,C 180,E1 -3015.761,E2 -3015.761} C_VEL
LIN {X 0,Y 559.169,Z 370.83,A -85,B 0,C 180,E1 -3018.23,E2 -3018.23} C_VEL
LIN {X 0,Y 559.181,Z 370.829,A -85,B 0,C 180,E1 -3021.191,E2 -3021.191} C_VEL
LIN {X 0,Y 559.16,Z 370.836,A -85,B 0,C 180,E1 -3023.791,E2 -3023.791} C_VEL
LIN {X 0,Y 559.166,Z 370.831,A -85,B 0,C 180,E1 -3026.425,E2 -3026.425} C_VEL
LIN {X 0,Y 559.16,Z 370.837,A -85,B 0,C 180,E1 -3028.981,E2 -3028.981} C_VEL
LIN {X 0,Y 559.172,Z 370.829,A -85,B 0,C 180,E1 -3031.619,E2 -3031.619} C_VEL
LIN {X 0,Y 559.185,Z 370.83,A -85,B 0,C 180,E1 -3033.903,E2 -3033.903} C_VEL
LIN {X 0,Y 559.143,Z 370.834,A -85,B 0,C 180,E1 -3036.572,E2 -3036.572} C_VEL
LIN {X 0,Y 559.184,Z 370.834,A -85,B 0,C 180,E1 -3039.396,E2 -3039.396} C_VEL
LIN {X 0,Y 559.15,Z 370.833,A -85,B 0,C 180,E1 -3041.686,E2 -3041.686} C_VEL
LIN {X 0,Y 559.17,Z 370.83,A -85,B 0,C 180,E1 -3043.948,E2 -3043.948} C_VEL
LIN {X 0,Y 559.178,Z 370.834,A -85,B 0,C 180,E1 -3046.184,E2 -3046.184} C_VEL
LIN {X 0,Y 559.197,Z 370.828,A -85,B 0,C 180,E1 -3049.134,E2 -3049.134} C_VEL
LIN {X 0,Y 559.21,Z 370.826,A -85,B 0,C 180,E1 -3052.054,E2 -3052.054} C_VEL
LIN {X 0,Y 559.257,Z 370.823,A -85,B 0,C 180,E1 -3054.953,E2 -3054.953} C_VEL
LIN {X 0,Y 559.256,Z 370.821,A -85,B 0,C 180,E1 -3057.839,E2 -3057.839} C_VEL
LIN {X 0,Y 559.276,Z 370.817,A -85,B 0,C 180,E1 -3060.72,E2 -3060.72} C_VEL
LIN {X 0,Y 559.242,Z 370.823,A -85,B 0,C 180,E1 -3062.881,E2 -3062.881} C_VEL
LIN {X 0,Y 559.231,Z 370.823,A -85,B 0,C 180,E1 -3065.77,E2 -3065.77} C_VEL
LIN {X 0,Y 559.176,Z 370.833,A -85,B 0,C 180,E1 -3068.675,E2 -3068.675} C_VEL
LIN {X 0,Y 559.21,Z 370.827,A -85,B 0,C 180,E1 -3071.6,E2 -3071.6} C_VEL
LIN {X 0,Y 559.205,Z 370.826,A -85,B 0,C 180,E1 -3074.596,E2 -3074.596} C_VEL
LIN {X 0,Y 559.145,Z 370.835,A -85,B 0,C 180,E1 -3077.557,E2 -3077.557} C_VEL
LIN {X 0,Y 559.178,Z 370.83,A -85,B 0,C 180,E1 -3079.837,E2 -3079.837} C_VEL
LIN {X 0,Y 559.145,Z 370.84,A -85,B 0,C 180,E1 -3082.153,E2 -3082.153} C_VEL
LIN {X 0,Y 559.18,Z 370.831,A -85,B 0,C 180,E1 -3085.298,E2 -3085.298} C_VEL
LIN {X 0,Y 559.185,Z 370.831,A -85,B 0,C 180,E1 -3087.712,E2 -3087.712} C_VEL
LIN {X 0,Y 559.144,Z 370.834,A -85,B 0,C 180,E1 -3090.618,E2 -3090.618} C_VEL
LIN {X 0,Y 558.482,Z 370.919,A -85,B 0,C 180,E1 -3091.219,E2 -3091.219} C_VEL
LIN {X 0,Y 555.62,Z 371.276,A -85,B 0,C 180,E1 -3092.195,E2 -3092.195} C_VEL
LIN {X 0,Y 553.207,Z 371.574,A -85,B 0,C 180,E1 -3092.981,E2 -3092.981} C_VEL
LIN {X 0,Y 552.188,Z 371.701,A -85,B 0,C 180,E1 -3093.587,E2 -3093.587} C_VEL
LIN {X 0,Y 552.114,Z 371.711,A -85,B 0,C 180,E1 -3093.793,E2 -3093.793} C_VEL
LIN {X 0,Y 552.109,Z 371.709,A -85,B 0,C 180,E1 -3096.747,E2 -3096.747} C_VEL
LIN {X 0,Y 552.136,Z 371.71,A -85,B 0,C 180,E1 -3099.527,E2 -3099.527} C_VEL
LIN {X 0,Y 552.133,Z 371.71,A -85,B 0,C 180,E1 -3102.425,E2 -3102.425} C_VEL
LIN {X 0,Y 552.102,Z 371.711,A -85,B 0,C 180,E1 -3105.563,E2 -3105.563} C_VEL
LIN {X 0,Y 552.134,Z 371.706,A -85,B 0,C 180,E1 -3108.677,E2 -3108.677} C_VEL
LIN {X 0,Y 552.121,Z 371.713,A -85,B 0,C 180,E1 -3111.411,E2 -3111.411} C_VEL
LIN {X 0,Y 552.06,Z 371.717,A -85,B 0,C 180,E1 -3114.154,E2 -3114.154} C_VEL
LIN {X 0,Y 551.94,Z 371.737,A -85,B 0,C 180,E1 -3115.926,E2 -3115.926} C_VEL
LIN {X 0,Y 551.894,Z 374.505,A -85,B 0,C 180,E1 -3118.562,E2 -3118.562} C_VEL
LIN {X 0,Y 551.874,Z 377.132,A -85,B 0,C 180,E1 -3121.058,E2 -3121.058} C_VEL
LIN {X 0,Y 551.84,Z 379.806,A -85,B 0,C 180,E1 -3123.529,E2 -3123.529} C_VEL
LIN {X 0,Y 551.792,Z 382.47,A -85,B 0,C 180,E1 -3125.947,E2 -3125.947} C_VEL
LIN {X 0,Y 551.726,Z 386.024,A -85,B 0,C 180,E1 -3129.104,E2 -3129.104} C_VEL
LIN {X 0,Y 551.676,Z 388.619,A -85,B 0,C 180,E1 -3131.429,E2 -3131.429} C_VEL
LIN {X 0,Y 551.707,Z 391.379,A -85,B 0,C 180,E1 -3133.725,E2 -3133.725} C_VEL
LIN {X 0,Y 551.702,Z 394.261,A -85,B 0,C 180,E1 -3135.993,E2 -3135.993} C_VEL
LIN {X 0,Y 551.71,Z 395.673,A -85,B 0,C 180,E1 -3137.096,E2 -3137.096} C_VEL
LIN {X 0,Y 553.029,Z 404.238,A -85,B 0,C 180,E1 -3137.337,E2 -3137.337} C_VEL
LIN {X 0,Y 552.896,Z 417.013,A -85,B 0,C 180,E1 -3137.753,E2 -3137.753} C_VEL
LIN {X 0,Y 552.723,Z 429.656,A -85,B 0,C 180,E1 -3138.332,E2 -3138.332} C_VEL
LIN {X 0,Y 552.53,Z 440.907,A -85,B 0,C 180,E1 -3139.001,E2 -3139.001} C_VEL
LIN {X 0,Y 552.336,Z 451.949,A -85,B 0,C 180,E1 -3139.831,E2 -3139.831} C_VEL
LIN {X 0,Y 552.153,Z 462.681,A -85,B 0,C 180,E1 -3140.845,E2 -3140.845} C_VEL
LIN {X 0,Y 552.007,Z 470.6,A -85,B 0,C 180,E1 -3141.765,E2 -3141.765} C_VEL
LIN {X 0,Y 551.895,Z 478.46,A -85,B 0,C 180,E1 -3142.886,E2 -3142.886} C_VEL
LIN {X 0,Y 551.868,Z 485.457,A -85,B 0,C 180,E1 -3144.153,E2 -3144.153} C_VEL
LIN {X 0,Y 551.725,Z 490.197,A -85,B 0,C 180,E1 -3145.251,E2 -3145.251} C_VEL
LIN {X 0,Y 551.751,Z 493.83,A -85,B 0,C 180,E1 -3146.349,E2 -3146.349} C_VEL
LIN {X 0,Y 551.723,Z 495.706,A -85,B 0,C 180,E1 -3147.079,E2 -3147.079} C_VEL
LIN {X 0,Y 551.657,Z 497.129,A -85,B 0,C 180,E1 -3147.81,E2 -3147.81} C_VEL
LIN {X 0,Y 551.642,Z 498.757,A -85,B 0,C 180,E1 -3149.27,E2 -3149.27} C_VEL
LIN {X 0,Y 551.641,Z 498.996,A -85,B 0,C 180,E1 -3150,E2 -3150} C_VEL
LIN {X 0,Y 551.641,Z 498.814,A -85,B 0,C 180,E1 -3150.73,E2 -3150.73} C_VEL
LIN {X 0,Y 551.657,Z 497.265,A -85,B 0,C 180,E1 -3152.19,E2 -3152.19} C_VEL
LIN {X 0,Y 551.724,Z 495.903,A -85,B 0,C 180,E1 -3152.921,E2 -3152.921} C_VEL
LIN {X 0,Y 551.764,Z 493.026,A -85,B 0,C 180,E1 -3154.017,E2 -3154.017} C_VEL
LIN {X 0,Y 551.723,Z 489.124,A -85,B 0,C 180,E1 -3155.116,E2 -3155.116} C_VEL
LIN {X 0,Y 551.811,Z 483.393,A -85,B 0,C 180,E1 -3156.349,E2 -3156.349} C_VEL
LIN {X 0,Y 551.925,Z 476.536,A -85,B 0,C 180,E1 -3157.5,E2 -3157.5} C_VEL
LIN {X 0,Y 552.063,Z 468.353,A -85,B 0,C 180,E1 -3158.603,E2 -3158.603} C_VEL
LIN {X 0,Y 552.198,Z 459.985,A -85,B 0,C 180,E1 -3159.524,E2 -3159.524} C_VEL
LIN {X 0,Y 552.414,Z 449.663,A -85,B 0,C 180,E1 -3160.445,E2 -3160.445} C_VEL
LIN {X 0,Y 552.572,Z 438.985,A -85,B 0,C 180,E1 -3161.214,E2 -3161.214} C_VEL
LIN {X 0,Y 552.739,Z 428.259,A -85,B 0,C 180,E1 -3161.831,E2 -3161.831} C_VEL
LIN {X 0,Y 552.878,Z 415.723,A -85,B 0,C 180,E1 -3162.387,E2 -3162.387} C_VEL
LIN {X 0,Y 552.911,Z 402.737,A -85,B 0,C 180,E1 -3162.794,E2 -3162.794} C_VEL
LIN {X 0,Y 551.695,Z 395.668,A -85,B 0,C 180,E1 -3162.998,E2 -3162.998} C_VEL
LIN {X 0,Y 551.669,Z 392.453,A -85,B 0,C 180,E1 -3165.518,E2 -3165.518} C_VEL
LIN {X 0,Y 551.685,Z 389.585,A -85,B 0,C 180,E1 -3167.803,E2 -3167.803} C_VEL
LIN {X 0,Y 551.726,Z 387.016,A -85,B 0,C 180,E1 -3170.117,E2 -3170.117} C_VEL
LIN {X 0,Y 551.766,Z 383.468,A -85,B 0,C 180,E1 -3173.257,E2 -3173.257} C_VEL
LIN {X 0,Y 551.822,Z 380.795,A -85,B 0,C 180,E1 -3175.66,E2 -3175.66} C_VEL
LIN {X 0,Y 551.869,Z 377.697,A -85,B 0,C 180,E1 -3178.513,E2 -3178.513} C_VEL
LIN {X 0,Y 551.906,Z 375.456,A -85,B 0,C 180,E1 -3180.622,E2 -3180.622} C_VEL
LIN {X 0,Y 551.918,Z 372.751,A -85,B 0,C 180,E1 -3183.2,E2 -3183.2} C_VEL
LIN {X 0,Y 551.931,Z 371.739,A -85,B 0,C 180,E1 -3184.139,E2 -3184.139} C_VEL
LIN {X 0,Y 552.106,Z 371.713,A -85,B 0,C 180,E1 -3186.747,E2 -3186.747} C_VEL
LIN {X 0,Y 552.134,Z 371.706,A -85,B 0,C 180,E1 -3189.527,E2 -3189.527} C_VEL
LIN {X 0,Y 552.136,Z 371.711,A -85,B 0,C 180,E1 -3192.425,E2 -3192.425} C_VEL
LIN {X 0,Y 552.098,Z 371.716,A -85,B 0,C 180,E1 -3195.562,E2 -3195.562} C_VEL
LIN {X 0,Y 552.125,Z 371.709,A -85,B 0,C 180,E1 -3198.554,E2 -3198.554} C_VEL
LIN {X 0,Y 552.125,Z 371.708,A -85,B 0,C 180,E1 -3201.411,E2 -3201.411} C_VEL
LIN {X 0,Y 552.105,Z 371.716,A -85,B 0,C 180,E1 -3204.158,E2 -3204.158} C_VEL
LIN {X 0,Y 552.121,Z 371.708,A -85,B 0,C 180,E1 -3206.814,E2 -3206.814} C_VEL
LIN {X 0,Y 552.108,Z 371.715,A -85,B 0,C 180,E1 -3209.391,E2 -3209.391} C_VEL
LIN {X 0,Y 552.115,Z 371.709,A -85,B 0,C 180,E1 -3211.902,E2 -3211.902} C_VEL
LIN {X 0,Y 552.161,Z 371.707,A -85,B 0,C 180,E1 -3214.65,E2 -3214.65} C_VEL
LIN {X 0,Y 552.097,Z 371.713,A -85,B 0,C 180,E1 -3217.549,E2 -3217.549} C_VEL
LIN {X 0,Y 552.155,Z 371.704,A -85,B 0,C 180,E1 -3220.374,E2 -3220.374} C_VEL
LIN {X 0,Y 552.16,Z 371.708,A -85,B 0,C 180,E1 -3222.977,E2 -3222.977} C_VEL
LIN {X 0,Y 552.141,Z 371.708,A -85,B 0,C 180,E1 -3226.005,E2 -3226.005} C_VEL
LIN {X 0,Y 552.167,Z 371.702,A -85,B 0,C 180,E1 -3228.993,E2 -3228.993} C_VEL
LIN {X 0,Y 552.156,Z 371.706,A -85,B 0,C 180,E1 -3231.951,E2 -3231.951} C_VEL
LIN {X 0,Y 552.233,Z 371.699,A -85,B 0,C 180,E1 -3234.889,E2 -3234.889} C_VEL
LIN {X 0,Y 552.224,Z 371.696,A -85,B 0,C 180,E1 -3237.812,E2 -3237.812} C_VEL
LIN {X 0,Y 552.247,Z 371.693,A -85,B 0,C 180,E1 -3240.729,E2 -3240.729} C_VEL
LIN {X 0,Y 552.209,Z 371.697,A -85,B 0,C 180,E1 -3242.918,E2 -3242.918} C_VEL
LIN {X 0,Y 552.202,Z 371.699,A -85,B 0,C 180,E1 -3245.844,E2 -3245.844} C_VEL
LIN {X 0,Y 552.167,Z 371.708,A -85,B 0,C 180,E1 -3248.786,E2 -3248.786} C_VEL
LIN {X 0,Y 552.169,Z 371.705,A -85,B 0,C 180,E1 -3251.75,E2 -3251.75} C_VEL
LIN {X 0,Y 552.142,Z 371.705,A -85,B 0,C 180,E1 -3254.748,E2 -3254.748} C_VEL
LIN {X 0,Y 552.104,Z 371.711,A -85,B 0,C 180,E1 -3257.789,E2 -3257.789} C_VEL
LIN {X 0,Y 552.137,Z 371.707,A -85,B 0,C 180,E1 -3260.101,E2 -3260.101} C_VEL
LIN {X 0,Y 552.097,Z 371.716,A -85,B 0,C 180,E1 -3262.451,E2 -3262.451} C_VEL
LIN {X 0,Y 552.161,Z 371.705,A -85,B 0,C 180,E1 -3265.35,E2 -3265.35} C_VEL
LIN {X 0,Y 552.125,Z 371.707,A -85,B 0,C 180,E1 -3268.098,E2 -3268.098} C_VEL
LIN {X 0,Y 552.108,Z 371.712,A -85,B 0,C 180,E1 -3270.609,E2 -3270.609} C_VEL
LIN {X 0,Y 552.12,Z 371.709,A -85,B 0,C 180,E1 -3273.186,E2 -3273.186} C_VEL
LIN {X 0,Y 552.09,Z 371.717,A -85,B 0,C 180,E1 -3275.843,E2 -3275.843} C_VEL
LIN {X 0,Y 552.13,Z 371.709,A -85,B 0,C 180,E1 -3279.062,E2 -3279.062} C_VEL
LIN {X 0,Y 552.125,Z 371.712,A -85,B 0,C 180,E1 -3281.446,E2 -3281.446} C_VEL
LIN {X 0,Y 552.1,Z 371.717,A -85,B 0,C 180,E1 -3284.532,E2 -3284.532} C_VEL
LIN {X 0,Y 552.136,Z 371.709,A -85,B 0,C 180,E1 -3287.584,E2 -3287.584} C_VEL
LIN {X 0,Y 552.133,Z 371.709,A -85,B 0,C 180,E1 -3290.473,E2 -3290.473} C_VEL
LIN {X 0,Y 552.141,Z 371.842,A -85,B 0,C 180,E1 -3292.57,E2 -3292.57} C_VEL
LIN {X 0,Y 552.916,Z 377.189,A -85,B 0,C 180,E1 -3294.439,E2 -3294.439} C_VEL
LIN {X 0,Y 552.872,Z 385.018,A -85,B 0,C 180,E1 -3297.033,E2 -3297.033} C_VEL
LIN {X 0,Y 552.67,Z 393.785,A -85,B 0,C 180,E1 -3299.851,E2 -3299.851} C_VEL
LIN {X 0,Y 552.521,Z 403.609,A -85,B 0,C 180,E1 -3302.923,E2 -3302.923} C_VEL
LIN {X 0,Y 552.356,Z 413.633,A -85,B 0,C 180,E1 -3305.973,E2 -3305.973} C_VEL
LIN {X 0,Y 552.2,Z 422.9,A -85,B 0,C 180,E1 -3308.732,E2 -3308.732} C_VEL
LIN {X 0,Y 552.086,Z 432.167,A -85,B 0,C 180,E1 -3311.443,E2 -3311.443} C_VEL
LIN {X 0,Y 551.982,Z 442.759,A -85,B 0,C 180,E1 -3314.492,E2 -3314.492} C_VEL
LIN {X 0,Y 551.914,Z 451.53,A -85,B 0,C 180,E1 -3316.983,E2 -3316.983} C_VEL
LIN {X 0,Y 553.107,Z 459.502,A -85,B 0,C 180,E1 -3317.175,E2 -3317.175} C_VEL
LIN {X 0,Y 552.977,Z 471.872,A -85,B 0,C 180,E1 -3317.522,E2 -3317.522} C_VEL
LIN {X 0,Y 552.827,Z 483.507,A -85,B 0,C 180,E1 -3317.985,E2 -3317.985} C_VEL
LIN {X 0,Y 552.643,Z 495.109,A -85,B 0,C 180,E1 -3318.592,E2 -3318.592} C_VEL
LIN {X 0,Y 552.426,Z 506.745,A -85,B 0,C 180,E1 -3319.37,E2 -3319.37} C_VEL
LIN {X 0,Y 552.234,Z 517.6,A -85,B 0,C 180,E1 -3320.292,E2 -3320.292} C_VEL
LIN {X 0,Y 552.079,Z 526.412,A -85,B 0,C 180,E1 -3321.213,E2 -3321.213} C_VEL
LIN {X 0,Y 551.95,Z 535,A -85,B 0,C 180,E1 -3322.317,E2 -3322.317} C_VEL
LIN {X 0,Y 551.823,Z 541.867,A -85,B 0,C 180,E1 -3323.418,E2 -3323.418} C_VEL
LIN {X 0,Y 551.804,Z 547.365,A -85,B 0,C 180,E1 -3324.518,E2 -3324.518} C_VEL
LIN {X 0,Y 551.764,Z 551.677,A -85,B 0,C 180,E1 -3325.617,E2 -3325.617} C_VEL
LIN {X 0,Y 551.75,Z 553.957,A -85,B 0,C 180,E1 -3326.348,E2 -3326.348} C_VEL
LIN {X 0,Y 551.723,Z 555.808,A -85,B 0,C 180,E1 -3327.079,E2 -3327.079} C_VEL
LIN {X 0,Y 551.657,Z 557.199,A -85,B 0,C 180,E1 -3327.81,E2 -3327.81} C_VEL
LIN {X 0,Y 551.641,Z 558.785,A -85,B 0,C 180,E1 -3329.27,E2 -3329.27} C_VEL
LIN {X 0,Y 551.64,Z 559,A -85,B 0,C 180,E1 -3330,E2 -3330} C_VEL
LIN {X 0,Y 551.645,Z 558.186,A -85,B 0,C 180,E1 -3331.46,E2 -3331.46} C_VEL
LIN {X 0,Y 551.657,Z 557.2,A -85,B 0,C 180,E1 -3332.19,E2 -3332.19} C_VEL
LIN {X 0,Y 551.723,Z 555.81,A -85,B 0,C 180,E1 -3332.921,E2 -3332.921} C_VEL
LIN {X 0,Y 551.763,Z 552.896,A -85,B 0,C 180,E1 -3334.017,E2 -3334.017} C_VEL
LIN {X 0,Y 551.724,Z 548.949,A -85,B 0,C 180,E1 -3335.116,E2 -3335.116} C_VEL
LIN {X 0,Y 551.803,Z 543.19,A -85,B 0,C 180,E1 -3336.342,E2 -3336.342} C_VEL
LIN {X 0,Y 551.926,Z 536.237,A -85,B 0,C 180,E1 -3337.5,E2 -3337.5} C_VEL
LIN {X 0,Y 552.082,Z 527.99,A -85,B 0,C 180,E1 -3338.602,E2 -3338.602} C_VEL
LIN {X 0,Y 552.201,Z 519.538,A -85,B 0,C 180,E1 -3339.524,E2 -3339.524} C_VEL
LIN {X 0,Y 552.425,Z 509.096,A -85,B 0,C 180,E1 -3340.445,E2 -3340.445} C_VEL
LIN {X 0,Y 552.599,Z 498.294,A -85,B 0,C 180,E1 -3341.214,E2 -3341.214} C_VEL
LIN {X 0,Y 552.751,Z 487.411,A -85,B 0,C 180,E1 -3341.831,E2 -3341.831} C_VEL
LIN {X 0,Y 552.881,Z 475.763,A -85,B 0,C 180,E1 -3342.34,E2 -3342.34} C_VEL
LIN {X 0,Y 553.037,Z 462.349,A -85,B 0,C 180,E1 -3342.756,E2 -3342.756} C_VEL
LIN {X 0,Y 552.909,Z 457.8,A -85,B 0,C 180,E1 -3342.864,E2 -3342.864} C_VEL
LIN {X 0,Y 551.914,Z 451.53,A -85,B 0,C 180,E1 -3343.016,E2 -3343.016} C_VEL
LIN {X 0,Y 551.996,Z 441.435,A -85,B 0,C 180,E1 -3345.887,E2 -3345.887} C_VEL
LIN {X 0,Y 552.085,Z 430.844,A -85,B 0,C 180,E1 -3348.942,E2 -3348.942} C_VEL
LIN {X 0,Y 552.255,Z 420.254,A -85,B 0,C 180,E1 -3352.05,E2 -3352.05} C_VEL
LIN {X 0,Y 552.4,Z 410.985,A -85,B 0,C 180,E1 -3354.825,E2 -3354.825} C_VEL
LIN {X 0,Y 552.533,Z 401.718,A -85,B 0,C 180,E1 -3357.663,E2 -3357.663} C_VEL
LIN {X 0,Y 552.704,Z 392.451,A -85,B 0,C 180,E1 -3360.573,E2 -3360.573} C_VEL
LIN {X 0,Y 552.883,Z 384.507,A -85,B 0,C 180,E1 -3363.134,E2 -3363.134} C_VEL
LIN {X 0,Y 552.894,Z 376.532,A -85,B 0,C 180,E1 -3365.783,E2 -3365.783} C_VEL
LIN {X 0,Y 552.114,Z 371.714,A -85,B 0,C 180,E1 -3367.547,E2 -3367.547} C_VEL
LIN {X 0,Y 552.113,Z 371.715,A -85,B 0,C 180,E1 -3370.481,E2 -3370.481} C_VEL
LIN {X 0,Y 552.118,Z 371.715,A -85,B 0,C 180,E1 -3373.484,E2 -3373.484} C_VEL
LIN {X 0,Y 552.109,Z 371.71,A -85,B 0,C 180,E1 -3376.576,E2 -3376.576} C_VEL
LIN {X 0,Y 552.123,Z 371.708,A -85,B 0,C 180,E1 -3379.52,E2 -3379.52} C_VEL
LIN {X 0,Y 552.097,Z 371.717,A -85,B 0,C 180,E1 -3382.336,E2 -3382.336} C_VEL
LIN {X 0,Y 552.122,Z 371.709,A -85,B 0,C 180,E1 -3385.054,E2 -3385.054} C_VEL
LIN {X 0,Y 552.12,Z 371.712,A -85,B 0,C 180,E1 -3387.682,E2 -3387.682} C_VEL
LIN {X 0,Y 552.115,Z 371.709,A -85,B 0,C 180,E1 -3390.235,E2 -3390.235} C_VEL
LIN {X 0,Y 552.143,Z 371.707,A -85,B 0,C 180,E1 -3393,E2 -3393} C_VEL
LIN {X 0,Y 552.117,Z 371.709,A -85,B 0,C 180,E1 -3395.161,E2 -3395.161} C_VEL
LIN {X 0,Y 552.13,Z 371.708,A -85,B 0,C 180,E1 -3398.337,E2 -3398.337} C_VEL
LIN {X 0,Y 552.161,Z 371.705,A -85,B 0,C 180,E1 -3400.675,E2 -3400.675} C_VEL
LIN {X 0,Y 552.12,Z 371.707,A -85,B 0,C 180,E1 -3403.737,E2 -3403.737} C_VEL
LIN {X 0,Y 552.141,Z 371.709,A -85,B 0,C 180,E1 -3406.005,E2 -3406.005} C_VEL
LIN {X 0,Y 552.165,Z 371.703,A -85,B 0,C 180,E1 -3408.993,E2 -3408.993} C_VEL
LIN {X 0,Y 552.164,Z 371.704,A -85,B 0,C 180,E1 -3411.952,E2 -3411.952} C_VEL
LIN {X 0,Y 552.232,Z 371.699,A -85,B 0,C 180,E1 -3414.889,E2 -3414.889} C_VEL
LIN {X 0,Y 552.228,Z 371.696,A -85,B 0,C 180,E1 -3417.812,E2 -3417.812} C_VEL
LIN {X 0,Y 552.246,Z 371.693,A -85,B 0,C 180,E1 -3420.729,E2 -3420.729} C_VEL
LIN {X 0,Y 552.208,Z 371.699,A -85,B 0,C 180,E1 -3422.918,E2 -3422.918} C_VEL
LIN {X 0,Y 552.202,Z 371.698,A -85,B 0,C 180,E1 -3425.844,E2 -3425.844} C_VEL
LIN {X 0,Y 552.147,Z 371.707,A -85,B 0,C 180,E1 -3428.786,E2 -3428.786} C_VEL
LIN {X 0,Y 552.168,Z 371.706,A -85,B 0,C 180,E1 -3431.75,E2 -3431.75} C_VEL
LIN {X 0,Y 552.141,Z 371.707,A -85,B 0,C 180,E1 -3434.748,E2 -3434.748} C_VEL
LIN {X 0,Y 552.103,Z 371.711,A -85,B 0,C 180,E1 -3437.789,E2 -3437.789} C_VEL
LIN {X 0,Y 552.136,Z 371.709,A -85,B 0,C 180,E1 -3440.101,E2 -3440.101} C_VEL
LIN {X 0,Y 552.096,Z 371.714,A -85,B 0,C 180,E1 -3442.451,E2 -3442.451} C_VEL
LIN {X 0,Y 552.16,Z 371.706,A -85,B 0,C 180,E1 -3445.35,E2 -3445.35} C_VEL
LIN {X 0,Y 552.124,Z 371.708,A -85,B 0,C 180,E1 -3448.098,E2 -3448.098} C_VEL
LIN {X 0,Y 552.107,Z 371.716,A -85,B 0,C 180,E1 -3450.614,E2 -3450.614} C_VEL
LIN {X 0,Y 552.119,Z 371.708,A -85,B 0,C 180,E1 -3453.186,E2 -3453.186} C_VEL
LIN {X 0,Y 552.114,Z 371.711,A -85,B 0,C 180,E1 -3453.793,E2 -3453.793} C_VEL
LIN {X 0,Y 551.48,Z 371.794,A -85,B 0,C 180,E1 -3454.401,E2 -3454.401} C_VEL
LIN {X 0,Y 548.657,Z 372.143,A -85,B 0,C 180,E1 -3455.389,E2 -3455.389} C_VEL
LIN {X 0,Y 546.235,Z 372.443,A -85,B 0,C 180,E1 -3456.184,E2 -3456.184} C_VEL
LIN {X 0,Y 545.166,Z 372.574,A -85,B 0,C 180,E1 -3456.798,E2 -3456.798} C_VEL
LIN {X 0,Y 545.065,Z 372.587,A -85,B 0,C 180,E1 -3457.006,E2 -3457.006} C_VEL
LIN {X 0,Y 545.075,Z 372.586,A -85,B 0,C 180,E1 -3460.142,E2 -3460.142} C_VEL
LIN {X 0,Y 545.082,Z 372.588,A -85,B 0,C 180,E1 -3463.107,E2 -3463.107} C_VEL
LIN {X 0,Y 545.068,Z 372.591,A -85,B 0,C 180,E1 -3466.225,E2 -3466.225} C_VEL
LIN {X 0,Y 545.091,Z 372.583,A -85,B 0,C 180,E1 -3468.886,E2 -3468.886} C_VEL
LIN {X 0,Y 545.055,Z 372.59,A -85,B 0,C 180,E1 -3471.763,E2 -3471.763} C_VEL
LIN {X 0,Y 544.997,Z 372.598,A -85,B 0,C 180,E1 -3474.333,E2 -3474.333} C_VEL
LIN {X 0,Y 544.846,Z 372.81,A -85,B 0,C 180,E1 -3476.313,E2 -3476.313} C_VEL
LIN {X 0,Y 544.817,Z 375.564,A -85,B 0,C 180,E1 -3478.936,E2 -3478.936} C_VEL
LIN {X 0,Y 544.828,Z 378.253,A -85,B 0,C 180,E1 -3481.492,E2 -3481.492} C_VEL
LIN {X 0,Y 544.778,Z 381.569,A -85,B 0,C 180,E1 -3484.562,E2 -3484.562} C_VEL
LIN {X 0,Y 544.662,Z 384.483,A -85,B 0,C 180,E1 -3487.226,E2 -3487.226} C_VEL
LIN {X 0,Y 544.642,Z 387.185,A -85,B 0,C 180,E1 -3489.61,E2 -3489.61} C_VEL
LIN {X 0,Y 544.635,Z 390.67,A -85,B 0,C 180,E1 -3492.735,E2 -3492.735} C_VEL
LIN {X 0,Y 544.627,Z 394.262,A -85,B 0,C 180,E1 -3495.807,E2 -3495.807} C_VEL
LIN {X 0,Y 544.607,Z 395.673,A -85,B 0,C 180,E1 -3496.924,E2 -3496.924} C_VEL
LIN {X 0,Y 546.084,Z 405.171,A -85,B 0,C 180,E1 -3497.197,E2 -3497.197} C_VEL
LIN {X 0,Y 545.932,Z 418.155,A -85,B 0,C 180,E1 -3497.642,E2 -3497.642} C_VEL
LIN {X 0,Y 545.756,Z 430.297,A -85,B 0,C 180,E1 -3498.215,E2 -3498.215} C_VEL
LIN {X 0,Y 545.545,Z 440.917,A -85,B 0,C 180,E1 -3498.858,E2 -3498.858} C_VEL
LIN {X 0,Y 545.344,Z 451.954,A -85,B 0,C 180,E1 -3499.699,E2 -3499.699} C_VEL
LIN {X 0,Y 545.123,Z 462.686,A -85,B 0,C 180,E1 -3500.726,E2 -3500.726} C_VEL
LIN {X 0,Y 544.975,Z 470.604,A -85,B 0,C 180,E1 -3501.658,E2 -3501.658} C_VEL
LIN {X 0,Y 544.829,Z 478.352,A -85,B 0,C 180,E1 -3502.775,E2 -3502.775} C_VEL
LIN {X 0,Y 544.778,Z 485.46,A -85,B 0,C 180,E1 -3504.076,E2 -3504.076} C_VEL
LIN {X 0,Y 544.628,Z 490.2,A -85,B 0,C 180,E1 -3505.189,E2 -3505.189} C_VEL
LIN {X 0,Y 544.669,Z 493.831,A -85,B 0,C 180,E1 -3506.301,E2 -3506.301} C_VEL
LIN {X 0,Y 544.65,Z 495.708,A -85,B 0,C 180,E1 -3507.041,E2 -3507.041} C_VEL
LIN {X 0,Y 544.572,Z 497.129,A -85,B 0,C 180,E1 -3507.781,E2 -3507.781} C_VEL
LIN {X 0,Y 544.542,Z 498.757,A -85,B 0,C 180,E1 -3509.261,E2 -3509.261} C_VEL
LIN {X 0,Y 544.542,Z 498.996,A -85,B 0,C 180,E1 -3510,E2 -3510} C_VEL
LIN {X 0,Y 544.542,Z 498.814,A -85,B 0,C 180,E1 -3510.74,E2 -3510.74} C_VEL
LIN {X 0,Y 544.572,Z 497.263,A -85,B 0,C 180,E1 -3512.219,E2 -3512.219} C_VEL
LIN {X 0,Y 544.651,Z 495.902,A -85,B 0,C 180,E1 -3512.959,E2 -3512.959} C_VEL
LIN {X 0,Y 544.684,Z 493.024,A -85,B 0,C 180,E1 -3514.07,E2 -3514.07} C_VEL
LIN {X 0,Y 544.653,Z 489.122,A -85,B 0,C 180,E1 -3515.182,E2 -3515.182} C_VEL
LIN {X 0,Y 544.725,Z 483.896,A -85,B 0,C 180,E1 -3516.335,E2 -3516.335} C_VEL
LIN {X 0,Y 544.859,Z 476.532,A -85,B 0,C 180,E1 -3517.598,E2 -3517.598} C_VEL
LIN {X 0,Y 544.999,Z 468.349,A -85,B 0,C 180,E1 -3518.715,E2 -3518.715} C_VEL
LIN {X 0,Y 545.159,Z 459.979,A -85,B 0,C 180,E1 -3519.648,E2 -3519.648} C_VEL
LIN {X 0,Y 545.404,Z 449.654,A -85,B 0,C 180,E1 -3520.581,E2 -3520.581} C_VEL
LIN {X 0,Y 545.615,Z 438.274,A -85,B 0,C 180,E1 -3521.405,E2 -3521.405} C_VEL
LIN {X 0,Y 545.783,Z 426.43,A -85,B 0,C 180,E1 -3522.079,E2 -3522.079} C_VEL
LIN {X 0,Y 545.999,Z 414.409,A -85,B 0,C 180,E1 -3522.593,E2 -3522.593} C_VEL
LIN {X 0,Y 545.952,Z 403.546,A -85,B 0,C 180,E1 -3522.939,E2 -3522.939} C_VEL
LIN {X 0,Y 544.596,Z 395.667,A -85,B 0,C 180,E1 -3523.171,E2 -3523.171} C_VEL
LIN {X 0,Y 544.591,Z 392.525,A -85,B 0,C 180,E1 -3525.724,E2 -3525.724} C_VEL
LIN {X 0,Y 544.608,Z 389.911,A -85,B 0,C 180,E1 -3528.042,E2 -3528.042} C_VEL
LIN {X 0,Y 544.643,Z 387.316,A -85,B 0,C 180,E1 -3530.39,E2 -3530.39} C_VEL
LIN {X 0,Y 544.725,Z 383.639,A -85,B 0,C 180,E1 -3533.646,E2 -3533.646} C_VEL
LIN {X 0,Y 544.757,Z 381.03,A -85,B 0,C 180,E1 -3536.017,E2 -3536.017} C_VEL
LIN {X 0,Y 544.811,Z 378.156,A -85,B 0,C 180,E1 -3538.694,E2 -3538.694} C_VEL
LIN {X 0,Y 544.818,Z 375.672,A -85,B 0,C 180,E1 -3541.064,E2 -3541.064} C_VEL
LIN {X 0,Y 544.851,Z 372.914,A -85,B 0,C 180,E1 -3543.687,E2 -3543.687} C_VEL
LIN {X 0,Y 544.992,Z 372.6,A -85,B 0,C 180,E1 -3545.472,E2 -3545.472} C_VEL
LIN {X 0,Y 545.054,Z 372.589,A -85,B 0,C 180,E1 -3548.136,E2 -3548.136} C_VEL
LIN {X 0,Y 545.086,Z 372.591,A -85,B 0,C 180,E1 -3550.473,E2 -3550.473} C_VEL
LIN {X 0,Y 545.086,Z 372.584,A -85,B 0,C 180,E1 -3553.106,E2 -3553.106} C_VEL
LIN {X 0,Y 545.054,Z 372.59,A -85,B 0,C 180,E1 -3556.226,E2 -3556.226} C_VEL
LIN {X 0,Y 545.086,Z 372.59,A -85,B 0,C 180,E1 -3558.886,E2 -3558.886} C_VEL
LIN {X 0,Y 545.089,Z 372.589,A -85,B 0,C 180,E1 -3560.819,E2 -3560.819} C_VEL
LIN {X 0,Y 545.054,Z 372.588,A -85,B 0,C 180,E1 -3563.62,E2 -3563.62} C_VEL
LIN {X 0,Y 545.073,Z 372.588,A -85,B 0,C 180,E1 -3566.328,E2 -3566.328} C_VEL
LIN {X 0,Y 545.071,Z 372.589,A -85,B 0,C 180,E1 -3568.952,E2 -3568.952} C_VEL
LIN {X 0,Y 545.106,Z 372.584,A -85,B 0,C 180,E1 -3571.508,E2 -3571.508} C_VEL
LIN {X 0,Y 545.1,Z 372.588,A -85,B 0,C 180,E1 -3574.491,E2 -3574.491} C_VEL
LIN {X 0,Y 545.042,Z 372.589,A -85,B 0,C 180,E1 -3577.242,E2 -3577.242} C_VEL
LIN {X 0,Y 545.127,Z 372.58,A -85,B 0,C 180,E1 -3580.415,E2 -3580.415} C_VEL
LIN {X 0,Y 545.075,Z 372.588,A -85,B 0,C 180,E1 -3583.521,E2 -3583.521} C_VEL
LIN {X 0,Y 545.101,Z 372.584,A -85,B 0,C 180,E1 -3585.82,E2 -3585.82} C_VEL
LIN {X 0,Y 545.123,Z 372.579,A -85,B 0,C 180,E1 -3588.849,E2 -3588.849} C_VEL
LIN {X 0,Y 545.103,Z 372.586,A -85,B 0,C 180,E1 -3591.847,E2 -3591.847} C_VEL
LIN {X 0,Y 545.209,Z 372.574,A -85,B 0,C 180,E1 -3594.823,E2 -3594.823} C_VEL
LIN {X 0,Y 545.196,Z 372.572,A -85,B 0,C 180,E1 -3597.784,E2 -3597.784} C_VEL
LIN {X 0,Y 545.218,Z 372.568,A -85,B 0,C 180,E1 -3600.739,E2 -3600.739} C_VEL
LIN {X 0,Y 545.176,Z 372.573,A -85,B 0,C 180,E1 -3602.956,E2 -3602.956} C_VEL
LIN {X 0,Y 545.174,Z 372.574,A -85,B 0,C 180,E1 -3605.919,E2 -3605.919} C_VEL
LIN {X 0,Y 545.125,Z 372.584,A -85,B 0,C 180,E1 -3608.9,E2 -3608.9} C_VEL
LIN {X 0,Y 545.141,Z 372.583,A -85,B 0,C 180,E1 -3611.904,E2 -3611.904} C_VEL
LIN {X 0,Y 545.091,Z 372.584,A -85,B 0,C 180,E1 -3614.943,E2 -3614.943} C_VEL
LIN {X 0,Y 545.076,Z 372.585,A -85,B 0,C 180,E1 -3618.026,E2 -3618.026} C_VEL
LIN {X 0,Y 545.101,Z 372.586,A -85,B 0,C 180,E1 -3620.372,E2 -3620.372} C_VEL
LIN {X 0,Y 545.084,Z 372.587,A -85,B 0,C 180,E1 -3623.559,E2 -3623.559} C_VEL
LIN {X 0,Y 545.085,Z 372.588,A -85,B 0,C 180,E1 -3626,E2 -3626} C_VEL
LIN {X 0,Y 545.094,Z 372.584,A -85,B 0,C 180,E1 -3628.748,E2 -3628.748} C_VEL
LIN {X 0,Y 545.062,Z 372.587,A -85,B 0,C 180,E1 -3631.679,E2 -3631.679} C_VEL
LIN {X 0,Y 545.067,Z 372.591,A -85,B 0,C 180,E1 -3634.564,E2 -3634.564} C_VEL
LIN {X 0,Y 545.041,Z 372.592,A -85,B 0,C 180,E1 -3637.304,E2 -3637.304} C_VEL
LIN {X 0,Y 545.073,Z 372.586,A -85,B 0,C 180,E1 -3640.142,E2 -3640.142} C_VEL
LIN {X 0,Y 545.082,Z 372.59,A -85,B 0,C 180,E1 -3643.106,E2 -3643.106} C_VEL
LIN {X 0,Y 545.069,Z 372.593,A -85,B 0,C 180,E1 -3646.224,E2 -3646.224} C_VEL
LIN {X 0,Y 545.092,Z 372.585,A -85,B 0,C 180,E1 -3648.886,E2 -3648.886} C_VEL
LIN {X 0,Y 545.055,Z 372.594,A -85,B 0,C 180,E1 -3651.763,E2 -3651.763} C_VEL
LIN {X 0,Y 545.097,Z 372.728,A -85,B 0,C 180,E1 -3652.351,E2 -3652.351} C_VEL
LIN {X 0,Y 545.943,Z 377.944,A -85,B 0,C 180,E1 -3654.195,E2 -3654.195} C_VEL
LIN {X 0,Y 545.917,Z 385.747,A -85,B 0,C 180,E1 -3656.803,E2 -3656.803} C_VEL
LIN {X 0,Y 545.693,Z 394.462,A -85,B 0,C 180,E1 -3659.644,E2 -3659.644} C_VEL
LIN {X 0,Y 545.542,Z 404.209,A -85,B 0,C 180,E1 -3662.736,E2 -3662.736} C_VEL
LIN {X 0,Y 545.352,Z 413.633,A -85,B 0,C 180,E1 -3665.645,E2 -3665.645} C_VEL
LIN {X 0,Y 545.173,Z 423.063,A -85,B 0,C 180,E1 -3668.493,E2 -3668.493} C_VEL
LIN {X 0,Y 545.029,Z 432.167,A -85,B 0,C 180,E1 -3671.194,E2 -3671.194} C_VEL
LIN {X 0,Y 544.924,Z 442.759,A -85,B 0,C 180,E1 -3674.285,E2 -3674.285} C_VEL
LIN {X 0,Y 544.829,Z 451.53,A -85,B 0,C 180,E1 -3676.811,E2 -3676.811} C_VEL
LIN {X 0,Y 546.152,Z 460.516,A -85,B 0,C 180,E1 -3677.033,E2 -3677.033} C_VEL
LIN {X 0,Y 546.031,Z 473.173,A -85,B 0,C 180,E1 -3677.408,E2 -3677.408} C_VEL
LIN {X 0,Y 545.841,Z 485.483,A -85,B 0,C 180,E1 -3677.923,E2 -3677.923} C_VEL
LIN {X 0,Y 545.631,Z 497.528,A -85,B 0,C 180,E1 -3678.591,E2 -3678.591} C_VEL
LIN {X 0,Y 545.416,Z 509.096,A -85,B 0,C 180,E1 -3679.419,E2 -3679.419} C_VEL
LIN {X 0,Y 545.166,Z 519.537,A -85,B 0,C 180,E1 -3680.352,E2 -3680.352} C_VEL
LIN {X 0,Y 545.029,Z 527.989,A -85,B 0,C 180,E1 -3681.285,E2 -3681.285} C_VEL
LIN {X 0,Y 544.86,Z 536.237,A -85,B 0,C 180,E1 -3682.402,E2 -3682.402} C_VEL
LIN {X 0,Y 544.734,Z 543.616,A -85,B 0,C 180,E1 -3683.655,E2 -3683.655} C_VEL
LIN {X 0,Y 544.653,Z 548.949,A -85,B 0,C 180,E1 -3684.818,E2 -3684.818} C_VEL
LIN {X 0,Y 544.683,Z 552.895,A -85,B 0,C 180,E1 -3685.93,E2 -3685.93} C_VEL
LIN {X 0,Y 544.65,Z 555.808,A -85,B 0,C 180,E1 -3687.041,E2 -3687.041} C_VEL
LIN {X 0,Y 544.546,Z 558.185,A -85,B 0,C 180,E1 -3688.521,E2 -3688.521} C_VEL
LIN {X 0,Y 544.541,Z 559,A -85,B 0,C 180,E1 -3690,E2 -3690} C_VEL
LIN {X 0,Y 544.546,Z 558.186,A -85,B 0,C 180,E1 -3691.479,E2 -3691.479} C_VEL
LIN {X 0,Y 544.65,Z 555.81,A -85,B 0,C 180,E1 -3692.959,E2 -3692.959} C_VEL
LIN {X 0,Y 544.683,Z 552.896,A -85,B 0,C 180,E1 -3694.069,E2 -3694.069} C_VEL
LIN {X 0,Y 544.653,Z 548.949,A -85,B 0,C 180,E1 -3695.182,E2 -3695.182} C_VEL
LIN {X 0,Y 544.74,Z 543.704,A -85,B 0,C 180,E1 -3696.328,E2 -3696.328} C_VEL
LIN {X 0,Y 544.836,Z 537.469,A -85,B 0,C 180,E1 -3697.411,E2 -3697.411} C_VEL
LIN {X 0,Y 545.007,Z 529.478,A -85,B 0,C 180,E1 -3698.528,E2 -3698.528} C_VEL
LIN {X 0,Y 545.142,Z 521.336,A -85,B 0,C 180,E1 -3699.461,E2 -3699.461} C_VEL
LIN {X 0,Y 545.372,Z 511.401,A -85,B 0,C 180,E1 -3700.394,E2 -3700.394} C_VEL
LIN {X 0,Y 545.541,Z 501.586,A -85,B 0,C 180,E1 -3701.142,E2 -3701.142} C_VEL
LIN {X 0,Y 545.739,Z 489.178,A -85,B 0,C 180,E1 -3701.891,E2 -3701.891} C_VEL
LIN {X 0,Y 545.923,Z 476.981,A -85,B 0,C 180,E1 -3702.453,E2 -3702.453} C_VEL
LIN {X 0,Y 546.128,Z 464.176,A -85,B 0,C 180,E1 -3702.873,E2 -3702.873} C_VEL
LIN {X 0,Y 545.851,Z 457.67,A -85,B 0,C 180,E1 -3703.036,E2 -3703.036} C_VEL
LIN {X 0,Y 544.829,Z 451.53,A -85,B 0,C 180,E1 -3703.189,E2 -3703.189} C_VEL
LIN {X 0,Y 544.94,Z 441.435,A -85,B 0,C 180,E1 -3706.098,E2 -3706.098} C_VEL
LIN {X 0,Y 545.068,Z 430.844,A -85,B 0,C 180,E1 -3709.196,E2 -3709.196} C_VEL
LIN {X 0,Y 545.216,Z 421.577,A -85,B 0,C 180,E1 -3711.951,E2 -3711.951} C_VEL
LIN {X 0,Y 545.376,Z 412.309,A -85,B 0,C 180,E1 -3714.76,E2 -3714.76} C_VEL
LIN {X 0,Y 545.526,Z 403.042,A -85,B 0,C 180,E1 -3717.632,E2 -3717.632} C_VEL
LIN {X 0,Y 545.733,Z 393.585,A -85,B 0,C 180,E1 -3720.638,E2 -3720.638} C_VEL
LIN {X 0,Y 545.917,Z 385.747,A -85,B 0,C 180,E1 -3723.197,E2 -3723.197} C_VEL
LIN {X 0,Y 545.951,Z 377.933,A -85,B 0,C 180,E1 -3725.806,E2 -3725.806} C_VEL
LIN {X 0,Y 545.055,Z 372.594,A -85,B 0,C 180,E1 -3727.768,E2 -3727.768} C_VEL
LIN {X 0,Y 545.085,Z 372.591,A -85,B 0,C 180,E1 -3730.473,E2 -3730.473} C_VEL
LIN {X 0,Y 545.09,Z 372.587,A -85,B 0,C 180,E1 -3733.106,E2 -3733.106} C_VEL
LIN {X 0,Y 545.053,Z 372.588,A -85,B 0,C 180,E1 -3736.226,E2 -3736.226} C_VEL
LIN {X 0,Y 545.094,Z 372.59,A -85,B 0,C 180,E1 -3738.886,E2 -3738.886} C_VEL
LIN {X 0,Y 545.057,Z 372.589,A -85,B 0,C 180,E1 -3741.763,E2 -3741.763} C_VEL
LIN {X 0,Y 545.055,Z 372.59,A -85,B 0,C 180,E1 -3744.533,E2 -3744.533} C_VEL
LIN {X 0,Y 545.073,Z 372.591,A -85,B 0,C 180,E1 -3747.212,E2 -3747.212} C_VEL
LIN {X 0,Y 545.068,Z 372.586,A -85,B 0,C 180,E1 -3749.811,E2 -3749.811} C_VEL
LIN {X 0,Y 545.093,Z 372.587,A -85,B 0,C 180,E1 -3752.344,E2 -3752.344} C_VEL
LIN {X 0,Y 545.121,Z 372.581,A -85,B 0,C 180,E1 -3754.821,E2 -3754.821} C_VEL
LIN {X 0,Y 545.04,Z 372.592,A -85,B 0,C 180,E1 -3757.242,E2 -3757.242} C_VEL
LIN {X 0,Y 545.125,Z 372.58,A -85,B 0,C 180,E1 -3760.415,E2 -3760.415} C_VEL
LIN {X 0,Y 545.077,Z 372.585,A -85,B 0,C 180,E1 -3763.521,E2 -3763.521} C_VEL
LIN {X 0,Y 545.1,Z 372.584,A -85,B 0,C 180,E1 -3765.82,E2 -3765.82} C_VEL
LIN {X 0,Y 545.121,Z 372.58,A -85,B 0,C 180,E1 -3768.849,E2 -3768.849} C_VEL
LIN {X 0,Y 545.135,Z 372.58,A -85,B 0,C 180,E1 -3771.847,E2 -3771.847} C_VEL
LIN {X 0,Y 545.208,Z 372.575,A -85,B 0,C 180,E1 -3774.823,E2 -3774.823} C_VEL
LIN {X 0,Y 545.199,Z 372.571,A -85,B 0,C 180,E1 -3777.784,E2 -3777.784} C_VEL
LIN {X 0,Y 545.216,Z 372.568,A -85,B 0,C 180,E1 -3780.739,E2 -3780.739} C_VEL
LIN {X 0,Y 545.175,Z 372.576,A -85,B 0,C 180,E1 -3782.956,E2 -3782.956} C_VEL
LIN {X 0,Y 545.174,Z 372.574,A -85,B 0,C 180,E1 -3785.92,E2 -3785.92} C_VEL
LIN {X 0,Y 545.108,Z 372.583,A -85,B 0,C 180,E1 -3788.9,E2 -3788.9} C_VEL
LIN {X 0,Y 545.14,Z 372.584,A -85,B 0,C 180,E1 -3791.904,E2 -3791.904} C_VEL
LIN {X 0,Y 545.09,Z 372.587,A -85,B 0,C 180,E1 -3794.944,E2 -3794.944} C_VEL
LIN {X 0,Y 545.075,Z 372.586,A -85,B 0,C 180,E1 -3798.026,E2 -3798.026} C_VEL
LIN {X 0,Y 545.101,Z 372.589,A -85,B 0,C 180,E1 -3800.372,E2 -3800.372} C_VEL
LIN {X 0,Y 545.084,Z 372.586,A -85,B 0,C 180,E1 -3803.559,E2 -3803.559} C_VEL
LIN {X 0,Y 545.084,Z 372.587,A -85,B 0,C 180,E1 -3806,E2 -3806} C_VEL
LIN {X 0,Y 545.093,Z 372.587,A -85,B 0,C 180,E1 -3808.748,E2 -3808.748} C_VEL
LIN {X 0,Y 545.062,Z 372.588,A -85,B 0,C 180,E1 -3811.679,E2 -3811.679} C_VEL
LIN {X 0,Y 545.067,Z 372.588,A -85,B 0,C 180,E1 -3814.564,E2 -3814.564} C_VEL
LIN {X 0,Y 545.065,Z 372.587,A -85,B 0,C 180,E1 -3817.006,E2 -3817.006} C_VEL
LIN {X 0,Y 544.359,Z 372.682,A -85,B 0,C 180,E1 -3817.623,E2 -3817.623} C_VEL
LIN {X 0,Y 541.496,Z 373.034,A -85,B 0,C 180,E1 -3818.624,E2 -3818.624} C_VEL
LIN {X 0,Y 539.11,Z 373.335,A -85,B 0,C 180,E1 -3819.429,E2 -3819.429} C_VEL
LIN {X 0,Y 538.1,Z 373.456,A -85,B 0,C 180,E1 -3820.052,E2 -3820.052} C_VEL
LIN {X 0,Y 538.024,Z 373.465,A -85,B 0,C 180,E1 -3820.262,E2 -3820.262} C_VEL
LIN {X 0,Y 538.03,Z 373.468,A -85,B 0,C 180,E1 -3822.988,E2 -3822.988} C_VEL
LIN {X 0,Y 538.022,Z 373.469,A -85,B 0,C 180,E1 -3826.186,E2 -3826.186} C_VEL
LIN {X 0,Y 538.053,Z 373.463,A -85,B 0,C 180,E1 -3829.253,E2 -3829.253} C_VEL
LIN {X 0,Y 537.995,Z 373.468,A -85,B 0,C 180,E1 -3832.122,E2 -3832.122} C_VEL
LIN {X 0,Y 537.93,Z 373.481,A -85,B 0,C 180,E1 -3834.91,E2 -3834.91} C_VEL
LIN {X 0,Y 537.839,Z 373.494,A -85,B 0,C 180,E1 -3835.814,E2 -3835.814} C_VEL
LIN {X 0,Y 537.783,Z 373.968,A -85,B 0,C 180,E1 -3836.76,E2 -3836.76} C_VEL
LIN {X 0,Y 537.782,Z 376.923,A -85,B 0,C 180,E1 -3839.601,E2 -3839.601} C_VEL
LIN {X 0,Y 537.723,Z 380.269,A -85,B 0,C 180,E1 -3842.777,E2 -3842.777} C_VEL
LIN {X 0,Y 537.675,Z 382.963,A -85,B 0,C 180,E1 -3845.274,E2 -3845.274} C_VEL
LIN {X 0,Y 537.606,Z 386.543,A -85,B 0,C 180,E1 -3848.528,E2 -3848.528} C_VEL
LIN {X 0,Y 537.555,Z 389.243,A -85,B 0,C 180,E1 -3850.922,E2 -3850.922} C_VEL
LIN {X 0,Y 537.553,Z 391.903,A -85,B 0,C 180,E1 -3853.284,E2 -3853.284} C_VEL
LIN {X 0,Y 537.516,Z 395.401,A -85,B 0,C 180,E1 -3856.388,E2 -3856.388} C_VEL
LIN {X 0,Y 537.522,Z 395.811,A -85,B 0,C 180,E1 -3856.749,E2 -3856.749} C_VEL
LIN {X 0,Y 539.144,Z 406.018,A -85,B 0,C 180,E1 -3857.053,E2 -3857.053} C_VEL
LIN {X 0,Y 538.966,Z 419.297,A -85,B 0,C 180,E1 -3857.527,E2 -3857.527} C_VEL
LIN {X 0,Y 538.787,Z 431.4,A -85,B 0,C 180,E1 -3858.119,E2 -3858.119} C_VEL
LIN {X 0,Y 538.547,Z 442.293,A -85,B 0,C 180,E1 -3858.807,E2 -3858.807} C_VEL
LIN {X 0,Y 538.319,Z 453.029,A -85,B 0,C 180,E1 -3859.659,E2 -3859.659} C_VEL
LIN {X 0,Y 538.087,Z 462.691,A -85,B 0,C 180,E1 -3860.604,E2 -3860.604} C_VEL
LIN {X 0,Y 537.923,Z 470.609,A -85,B 0,C 180,E1 -3861.548,E2 -3861.548} C_VEL
LIN {X 0,Y 537.76,Z 478.356,A -85,B 0,C 180,E1 -3862.679,E2 -3862.679} C_VEL
LIN {X 0,Y 537.694,Z 485.463,A -85,B 0,C 180,E1 -3863.998,E2 -3863.998} C_VEL
LIN {X 0,Y 537.54,Z 490.202,A -85,B 0,C 180,E1 -3865.125,E2 -3865.125} C_VEL
LIN {X 0,Y 537.591,Z 493.833,A -85,B 0,C 180,E1 -3866.252,E2 -3866.252} C_VEL
LIN {X 0,Y 537.551,Z 495.709,A -85,B 0,C 180,E1 -3867.002,E2 -3867.002} C_VEL
LIN {X 0,Y 537.49,Z 497.129,A -85,B 0,C 180,E1 -3867.752,E2 -3867.752} C_VEL
LIN {X 0,Y 537.442,Z 498.757,A -85,B 0,C 180,E1 -3869.251,E2 -3869.251} C_VEL
LIN {X 0,Y 537.442,Z 498.996,A -85,B 0,C 180,E1 -3870,E2 -3870} C_VEL
LIN {X 0,Y 537.442,Z 498.814,A -85,B 0,C 180,E1 -3870.749,E2 -3870.749} C_VEL
LIN {X 0,Y 537.49,Z 497.261,A -85,B 0,C 180,E1 -3872.248,E2 -3872.248} C_VEL
LIN {X 0,Y 537.552,Z 495.9,A -85,B 0,C 180,E1 -3872.998,E2 -3872.998} C_VEL
LIN {X 0,Y 537.604,Z 493.022,A -85,B 0,C 180,E1 -3874.123,E2 -3874.123} C_VEL
LIN {X 0,Y 537.587,Z 489.119,A -85,B 0,C 180,E1 -3875.251,E2 -3875.251} C_VEL
LIN {X 0,Y 537.639,Z 484.367,A -85,B 0,C 180,E1 -3876.321,E2 -3876.321} C_VEL
LIN {X 0,Y 537.79,Z 477.755,A -85,B 0,C 180,E1 -3877.509,E2 -3877.509} C_VEL
LIN {X 0,Y 537.952,Z 469.829,A -85,B 0,C 180,E1 -3878.641,E2 -3878.641} C_VEL
LIN {X 0,Y 538.13,Z 459.972,A -85,B 0,C 180,E1 -3879.775,E2 -3879.775} C_VEL
LIN {X 0,Y 538.377,Z 449.645,A -85,B 0,C 180,E1 -3880.721,E2 -3880.721} C_VEL
LIN {X 0,Y 538.636,Z 438.674,A -85,B 0,C 180,E1 -3881.527,E2 -3881.527} C_VEL
LIN {X 0,Y 538.813,Z 428.234,A -85,B 0,C 180,E1 -3882.142,E2 -3882.142} C_VEL
LIN {X 0,Y 539.022,Z 415.692,A -85,B 0,C 180,E1 -3882.711,E2 -3882.711} C_VEL
LIN {X 0,Y 538.956,Z 404.084,A -85,B 0,C 180,E1 -3883.095,E2 -3883.095} C_VEL
LIN {X 0,Y 537.526,Z 395.817,A -85,B 0,C 180,E1 -3883.347,E2 -3883.347} C_VEL
LIN {X 0,Y 537.536,Z 392.88,A -85,B 0,C 180,E1 -3885.936,E2 -3885.936} C_VEL
LIN {X 0,Y 537.543,Z 390.236,A -85,B 0,C 180,E1 -3888.288,E2 -3888.288} C_VEL
LIN {X 0,Y 537.56,Z 387.566,A -85,B 0,C 180,E1 -3890.671,E2 -3890.671} C_VEL
LIN {X 0,Y 537.648,Z 384.078,A -85,B 0,C 180,E1 -3893.79,E2 -3893.79} C_VEL
LIN {X 0,Y 537.689,Z 381.257,A -85,B 0,C 180,E1 -3896.386,E2 -3896.386} C_VEL
LIN {X 0,Y 537.745,Z 378.574,A -85,B 0,C 180,E1 -3898.919,E2 -3898.919} C_VEL
LIN {X 0,Y 537.774,Z 375.866,A -85,B 0,C 180,E1 -3901.517,E2 -3901.517} C_VEL
LIN {X 0,Y 537.784,Z 374.018,A -85,B 0,C 180,E1 -3903.29,E2 -3903.29} C_VEL
LIN {X 0,Y 537.889,Z 373.488,A -85,B 0,C 180,E1 -3904.598,E2 -3904.598} C_VEL
LIN {X 0,Y 538.007,Z 373.471,A -85,B 0,C 180,E1 -3907.17,E2 -3907.17} C_VEL
LIN {X 0,Y 538.027,Z 373.463,A -85,B 0,C 180,E1 -3909.797,E2 -3909.797} C_VEL
LIN {X 0,Y 538.026,Z 373.465,A -85,B 0,C 180,E1 -3912.786,E2 -3912.786} C_VEL
LIN {X 0,Y 538.012,Z 373.467,A -85,B 0,C 180,E1 -3915.138,E2 -3915.138} C_VEL
LIN {X 0,Y 538.035,Z 373.464,A -85,B 0,C 180,E1 -3918.227,E2 -3918.227} C_VEL
LIN {X 0,Y 538.021,Z 373.467,A -85,B 0,C 180,E1 -3921.17,E2 -3921.17} C_VEL
LIN {X 0,Y 538.028,Z 373.468,A -85,B 0,C 180,E1 -3924.084,E2 -3924.084} C_VEL
LIN {X 0,Y 538.035,Z 373.463,A -85,B 0,C 180,E1 -3926.728,E2 -3926.728} C_VEL
LIN {X 0,Y 538.031,Z 373.468,A -85,B 0,C 180,E1 -3929.556,E2 -3929.556} C_VEL
LIN {X 0,Y 538.045,Z 373.462,A -85,B 0,C 180,E1 -3931.95,E2 -3931.95} C_VEL
LIN {X 0,Y 538.076,Z 373.463,A -85,B 0,C 180,E1 -3934.467,E2 -3934.467} C_VEL
LIN {X 0,Y 537.998,Z 373.471,A -85,B 0,C 180,E1 -3937.738,E2 -3937.738} C_VEL
LIN {X 0,Y 538.085,Z 373.458,A -85,B 0,C 180,E1 -3940.148,E2 -3940.148} C_VEL
LIN {X 0,Y 538.023,Z 373.468,A -85,B 0,C 180,E1 -3943.299,E2 -3943.299} C_VEL
LIN {X 0,Y 538.07,Z 373.459,A -85,B 0,C 180,E1 -3945.631,E2 -3945.631} C_VEL
LIN {X 0,Y 538.083,Z 373.457,A -85,B 0,C 180,E1 -3948.702,E2 -3948.702} C_VEL
LIN {X 0,Y 538.067,Z 373.463,A -85,B 0,C 180,E1 -3951.739,E2 -3951.739} C_VEL
LIN {X 0,Y 538.128,Z 373.452,A -85,B 0,C 180,E1 -3954.003,E2 -3954.003} C_VEL
LIN {X 0,Y 538.142,Z 373.453,A -85,B 0,C 180,E1 -3957.006,E2 -3957.006} C_VEL
LIN {X 0,Y 538.178,Z 373.451,A -85,B 0,C 180,E1 -3960,E2 -3960} C_VEL
LIN {X 0,Y 538.142,Z 373.449,A -85,B 0,C 180,E1 -3962.994,E2 -3962.994} C_VEL
LIN {X 0,Y 538.128,Z 373.452,A -85,B 0,C 180,E1 -3965.997,E2 -3965.997} C_VEL
LIN {X 0,Y 538.076,Z 373.461,A -85,B 0,C 180,E1 -3969.018,E2 -3969.018} C_VEL
LIN {X 0,Y 538.089,Z 373.461,A -85,B 0,C 180,E1 -3972.062,E2 -3972.062} C_VEL
LIN {X 0,Y 538.05,Z 373.463,A -85,B 0,C 180,E1 -3975.144,E2 -3975.144} C_VEL
LIN {X 0,Y 538.031,Z 373.463,A -85,B 0,C 180,E1 -3978.27,E2 -3978.27} C_VEL
LIN {X 0,Y 538.045,Z 373.466,A -85,B 0,C 180,E1 -3980.651,E2 -3980.651} C_VEL
LIN {X 0,Y 538.008,Z 373.472,A -85,B 0,C 180,E1 -3983.888,E2 -3983.888} C_VEL
LIN {X 0,Y 538.047,Z 373.462,A -85,B 0,C 180,E1 -3986.366,E2 -3986.366} C_VEL
LIN {X 0,Y 538.036,Z 373.465,A -85,B 0,C 180,E1 -3988.933,E2 -3988.933} C_VEL
LIN {X 0,Y 538.015,Z 373.466,A -85,B 0,C 180,E1 -3991.887,E2 -3991.887} C_VEL
LIN {X 0,Y 538.017,Z 373.469,A -85,B 0,C 180,E1 -3994.618,E2 -3994.618} C_VEL
LIN {X 0,Y 538.009,Z 373.467,A -85,B 0,C 180,E1 -3997.17,E2 -3997.17} C_VEL
LIN {X 0,Y 538.03,Z 373.466,A -85,B 0,C 180,E1 -3999.796,E2 -3999.796} C_VEL
LIN {X 0,Y 538.023,Z 373.471,A -85,B 0,C 180,E1 -4002.786,E2 -4002.786} C_VEL
LIN {X 0,Y 538.037,Z 373.464,A -85,B 0,C 180,E1 -4005.141,E2 -4005.141} C_VEL
LIN {X 0,Y 538.041,Z 373.467,A -85,B 0,C 180,E1 -4008.227,E2 -4008.227} C_VEL
LIN {X 0,Y 538.016,Z 373.471,A -85,B 0,C 180,E1 -4011.169,E2 -4011.169} C_VEL
LIN {X 0,Y 538.041,Z 373.58,A -85,B 0,C 180,E1 -4012.126,E2 -4012.126} C_VEL
LIN {X 0,Y 538.944,Z 378.988,A -85,B 0,C 180,E1 -4014.068,E2 -4014.068} C_VEL
LIN {X 0,Y 538.971,Z 385.498,A -85,B 0,C 180,E1 -4016.276,E2 -4016.276} C_VEL
LIN {X 0,Y 538.76,Z 393.774,A -85,B 0,C 180,E1 -4018.984,E2 -4018.984} C_VEL
LIN {X 0,Y 538.587,Z 403.041,A -85,B 0,C 180,E1 -4021.981,E2 -4021.981} C_VEL
LIN {X 0,Y 538.368,Z 412.309,A -85,B 0,C 180,E1 -4024.896,E2 -4024.896} C_VEL
LIN {X 0,Y 538.18,Z 422.407,A -85,B 0,C 180,E1 -4028,E2 -4028} C_VEL
LIN {X 0,Y 538.025,Z 430.844,A -85,B 0,C 180,E1 -4030.543,E2 -4030.543} C_VEL
LIN {X 0,Y 537.896,Z 440.111,A -85,B 0,C 180,E1 -4033.295,E2 -4033.295} C_VEL
LIN {X 0,Y 537.792,Z 449.378,A -85,B 0,C 180,E1 -4036.009,E2 -4036.009} C_VEL
LIN {X 0,Y 537.757,Z 451.53,A -85,B 0,C 180,E1 -4036.634,E2 -4036.634} C_VEL
LIN {X 0,Y 539.225,Z 461.431,A -85,B 0,C 180,E1 -4036.887,E2 -4036.887} C_VEL
LIN {X 0,Y 539.083,Z 474.47,A -85,B 0,C 180,E1 -4037.291,E2 -4037.291} C_VEL
LIN {X 0,Y 538.901,Z 485.484,A -85,B 0,C 180,E1 -4037.765,E2 -4037.765} C_VEL
LIN {X 0,Y 538.68,Z 496.274,A -85,B 0,C 180,E1 -4038.363,E2 -4038.363} C_VEL
LIN {X 0,Y 538.475,Z 506.744,A -85,B 0,C 180,E1 -4039.091,E2 -4039.091} C_VEL
LIN {X 0,Y 538.202,Z 517.6,A -85,B 0,C 180,E1 -4040.036,E2 -4040.036} C_VEL
LIN {X 0,Y 538.015,Z 526.412,A -85,B 0,C 180,E1 -4040.981,E2 -4040.981} C_VEL
LIN {X 0,Y 537.829,Z 535,A -85,B 0,C 180,E1 -4042.114,E2 -4042.114} C_VEL
LIN {X 0,Y 537.705,Z 541.867,A -85,B 0,C 180,E1 -4043.244,E2 -4043.244} C_VEL
LIN {X 0,Y 537.676,Z 547.365,A -85,B 0,C 180,E1 -4044.374,E2 -4044.374} C_VEL
LIN {X 0,Y 537.557,Z 551.677,A -85,B 0,C 180,E1 -4045.501,E2 -4045.501} C_VEL
LIN {X 0,Y 537.591,Z 553.957,A -85,B 0,C 180,E1 -4046.252,E2 -4046.252} C_VEL
LIN {X 0,Y 537.551,Z 555.808,A -85,B 0,C 180,E1 -4047.002,E2 -4047.002} C_VEL
LIN {X 0,Y 537.49,Z 557.198,A -85,B 0,C 180,E1 -4047.752,E2 -4047.752} C_VEL
LIN {X 0,Y 537.442,Z 558.785,A -85,B 0,C 180,E1 -4049.251,E2 -4049.251} C_VEL
LIN {X 0,Y 537.442,Z 559,A -85,B 0,C 180,E1 -4050,E2 -4050} C_VEL
LIN {X 0,Y 537.452,Z 558.186,A -85,B 0,C 180,E1 -4051.499,E2 -4051.499} C_VEL
LIN {X 0,Y 537.49,Z 557.199,A -85,B 0,C 180,E1 -4052.248,E2 -4052.248} C_VEL
LIN {X 0,Y 537.551,Z 555.81,A -85,B 0,C 180,E1 -4052.998,E2 -4052.998} C_VEL
LIN {X 0,Y 537.603,Z 552.896,A -85,B 0,C 180,E1 -4054.123,E2 -4054.123} C_VEL
LIN {X 0,Y 537.587,Z 548.949,A -85,B 0,C 180,E1 -4055.251,E2 -4055.251} C_VEL
LIN {X 0,Y 537.65,Z 544.079,A -85,B 0,C 180,E1 -4056.335,E2 -4056.335} C_VEL
LIN {X 0,Y 537.791,Z 537.469,A -85,B 0,C 180,E1 -4057.509,E2 -4057.509} C_VEL
LIN {X 0,Y 537.972,Z 529.478,A -85,B 0,C 180,E1 -4058.64,E2 -4058.64} C_VEL
LIN {X 0,Y 538.119,Z 521.336,A -85,B 0,C 180,E1 -4059.585,E2 -4059.585} C_VEL
LIN {X 0,Y 538.367,Z 511.401,A -85,B 0,C 180,E1 -4060.531,E2 -4060.531} C_VEL
LIN {X 0,Y 538.576,Z 501.587,A -85,B 0,C 180,E1 -4061.288,E2 -4061.288} C_VEL
LIN {X 0,Y 538.751,Z 490.55,A -85,B 0,C 180,E1 -4061.973,E2 -4061.973} C_VEL
LIN {X 0,Y 538.959,Z 478.11,A -85,B 0,C 180,E1 -4062.568,E2 -4062.568} C_VEL
LIN {X 0,Y 539.197,Z 465.089,A -85,B 0,C 180,E1 -4063.017,E2 -4063.017} C_VEL
LIN {X 0,Y 538.956,Z 458.793,A -85,B 0,C 180,E1 -4063.182,E2 -4063.182} C_VEL
LIN {X 0,Y 537.757,Z 451.53,A -85,B 0,C 180,E1 -4063.365,E2 -4063.365} C_VEL
LIN {X 0,Y 537.876,Z 442.759,A -85,B 0,C 180,E1 -4065.926,E2 -4065.926} C_VEL
LIN {X 0,Y 537.988,Z 433.492,A -85,B 0,C 180,E1 -4068.666,E2 -4068.666} C_VEL
LIN {X 0,Y 538.128,Z 424.225,A -85,B 0,C 180,E1 -4071.45,E2 -4071.45} C_VEL
LIN {X 0,Y 538.332,Z 414.958,A -85,B 0,C 180,E1 -4074.282,E2 -4074.282} C_VEL
LIN {X 0,Y 538.528,Z 404.842,A -85,B 0,C 180,E1 -4077.448,E2 -4077.448} C_VEL
LIN {X 0,Y 538.733,Z 395.099,A -85,B 0,C 180,E1 -4080.582,E2 -4080.582} C_VEL
LIN {X 0,Y 538.967,Z 386.363,A -85,B 0,C 180,E1 -4083.431,E2 -4083.431} C_VEL
LIN {X 0,Y 539.031,Z 380.313,A -85,B 0,C 180,E1 -4085.465,E2 -4085.465} C_VEL
LIN {X 0,Y 538.384,Z 375.335,A -85,B 0,C 180,E1 -4087.223,E2 -4087.223} C_VEL
LIN {X 0,Y 538.006,Z 373.472,A -85,B 0,C 180,E1 -4088.005,E2 -4088.005} C_VEL
LIN {X 0,Y 538.052,Z 373.464,A -85,B 0,C 180,E1 -4090.776,E2 -4090.776} C_VEL
LIN {X 0,Y 538.033,Z 373.469,A -85,B 0,C 180,E1 -4094.075,E2 -4094.075} C_VEL
LIN {X 0,Y 538.022,Z 373.47,A -85,B 0,C 180,E1 -4097.214,E2 -4097.214} C_VEL
LIN {X 0,Y 538.031,Z 373.465,A -85,B 0,C 180,E1 -4100.204,E2 -4100.204} C_VEL
LIN {X 0,Y 538.03,Z 373.464,A -85,B 0,C 180,E1 -4103.067,E2 -4103.067} C_VEL
LIN {X 0,Y 538.028,Z 373.468,A -85,B 0,C 180,E1 -4105.827,E2 -4105.827} C_VEL
LIN {X 0,Y 538.012,Z 373.466,A -85,B 0,C 180,E1 -4108.499,E2 -4108.499} C_VEL
LIN {X 0,Y 538.064,Z 373.462,A -85,B 0,C 180,E1 -4111.1,E2 -4111.1} C_VEL
LIN {X 0,Y 538.046,Z 373.462,A -85,B 0,C 180,E1 -4113.633,E2 -4113.633} C_VEL
LIN {X 0,Y 538.011,Z 373.471,A -85,B 0,C 180,E1 -4116.122,E2 -4116.122} C_VEL
LIN {X 0,Y 538.044,Z 373.467,A -85,B 0,C 180,E1 -4119.349,E2 -4119.349} C_VEL
LIN {X 0,Y 538.059,Z 373.463,A -85,B 0,C 180,E1 -4122.517,E2 -4122.517} C_VEL
LIN {X 0,Y 538.069,Z 373.459,A -85,B 0,C 180,E1 -4125.631,E2 -4125.631} C_VEL
LIN {X 0,Y 538.081,Z 373.458,A -85,B 0,C 180,E1 -4128.702,E2 -4128.702} C_VEL
LIN {X 0,Y 538.092,Z 373.459,A -85,B 0,C 180,E1 -4131.74,E2 -4131.74} C_VEL
LIN {X 0,Y 538.165,Z 373.453,A -85,B 0,C 180,E1 -4134.755,E2 -4134.755} C_VEL
LIN {X 0,Y 538.171,Z 373.446,A -85,B 0,C 180,E1 -4137.755,E2 -4137.755} C_VEL
LIN {X 0,Y 538.186,Z 373.444,A -85,B 0,C 180,E1 -4140.748,E2 -4140.748} C_VEL
LIN {X 0,Y 538.141,Z 373.453,A -85,B 0,C 180,E1 -4142.994,E2 -4142.994} C_VEL
LIN {X 0,Y 538.127,Z 373.452,A -85,B 0,C 180,E1 -4145.997,E2 -4145.997} C_VEL
LIN {X 0,Y 538.06,Z 373.46,A -85,B 0,C 180,E1 -4149.018,E2 -4149.018} C_VEL
LIN {X 0,Y 538.088,Z 373.461,A -85,B 0,C 180,E1 -4152.062,E2 -4152.062} C_VEL
LIN {X 0,Y 538.05,Z 373.465,A -85,B 0,C 180,E1 -4155.144,E2 -4155.144} C_VEL
LIN {X 0,Y 538.03,Z 373.465,A -85,B 0,C 180,E1 -4158.27,E2 -4158.27} C_VEL
LIN {X 0,Y 538.044,Z 373.465,A -85,B 0,C 180,E1 -4160.651,E2 -4160.651} C_VEL
LIN {X 0,Y 538.007,Z 373.472,A -85,B 0,C 180,E1 -4163.888,E2 -4163.888} C_VEL
LIN {X 0,Y 538.046,Z 373.462,A -85,B 0,C 180,E1 -4166.367,E2 -4166.367} C_VEL
LIN {X 0,Y 538.035,Z 373.467,A -85,B 0,C 180,E1 -4168.933,E2 -4168.933} C_VEL
LIN {X 0,Y 538.014,Z 373.467,A -85,B 0,C 180,E1 -4171.887,E2 -4171.887} C_VEL
LIN {X 0,Y 538.016,Z 373.466,A -85,B 0,C 180,E1 -4174.618,E2 -4174.618} C_VEL
LIN {X 0,Y 538.008,Z 373.467,A -85,B 0,C 180,E1 -4177.17,E2 -4177.17} C_VEL
LIN {X 0,Y 538.024,Z 373.465,A -85,B 0,C 180,E1 -4180.262,E2 -4180.262} C_VEL
LIN {X 0,Y 537.373,Z 373.55,A -85,B 0,C 180,E1 -4180.887,E2 -4180.887} C_VEL
LIN {X 0,Y 534.52,Z 373.904,A -85,B 0,C 180,E1 -4181.902,E2 -4181.902} C_VEL
LIN {X 0,Y 532.092,Z 374.207,A -85,B 0,C 180,E1 -4182.719,E2 -4182.719} C_VEL
LIN {X 0,Y 531.043,Z 374.335,A -85,B 0,C 180,E1 -4183.35,E2 -4183.35} C_VEL
LIN {X 0,Y 530.955,Z 374.345,A -85,B 0,C 180,E1 -4183.564,E2 -4183.564} C_VEL
LIN {X 0,Y 530.97,Z 374.345,A -85,B 0,C 180,E1 -4186.506,E2 -4186.506} C_VEL
LIN {X 0,Y 530.99,Z 374.34,A -85,B 0,C 180,E1 -4188.976,E2 -4188.976} C_VEL
LIN {X 0,Y 530.961,Z 374.348,A -85,B 0,C 180,E1 -4191.529,E2 -4191.529} C_VEL
LIN {X 0,Y 530.91,Z 374.354,A -85,B 0,C 180,E1 -4194.376,E2 -4194.376} C_VEL
LIN {X 0,Y 530.73,Z 374.438,A -85,B 0,C 180,E1 -4196.539,E2 -4196.539} C_VEL
LIN {X 0,Y 530.696,Z 377.396,A -85,B 0,C 180,E1 -4199.406,E2 -4199.406} C_VEL
LIN {X 0,Y 530.661,Z 380.667,A -85,B 0,C 180,E1 -4202.541,E2 -4202.541} C_VEL
LIN {X 0,Y 530.599,Z 383.193,A -85,B 0,C 180,E1 -4204.922,E2 -4204.922} C_VEL
LIN {X 0,Y 530.545,Z 386.584,A -85,B 0,C 180,E1 -4208.014,E2 -4208.014} C_VEL
LIN {X 0,Y 530.509,Z 389.52,A -85,B 0,C 180,E1 -4210.659,E2 -4210.659} C_VEL
LIN {X 0,Y 530.489,Z 392.234,A -85,B 0,C 180,E1 -4213.055,E2 -4213.055} C_VEL
LIN {X 0,Y 530.442,Z 395.783,A -85,B 0,C 180,E1 -4216.203,E2 -4216.203} C_VEL
LIN {X 0,Y 530.463,Z 396.266,A -85,B 0,C 180,E1 -4216.582,E2 -4216.582} C_VEL
LIN {X 0,Y 532.257,Z 406.468,A -85,B 0,C 180,E1 -4216.883,E2 -4216.883} C_VEL
LIN {X 0,Y 532.051,Z 419.702,A -85,B 0,C 180,E1 -4217.363,E2 -4217.363} C_VEL
LIN {X 0,Y 531.863,Z 430.875,A -85,B 0,C 180,E1 -4217.914,E2 -4217.914} C_VEL
LIN {X 0,Y 531.596,Z 442.575,A -85,B 0,C 180,E1 -4218.659,E2 -4218.659} C_VEL
LIN {X 0,Y 531.328,Z 453.236,A -85,B 0,C 180,E1 -4219.521,E2 -4219.521} C_VEL
LIN {X 0,Y 531.072,Z 462.822,A -85,B 0,C 180,E1 -4220.478,E2 -4220.478} C_VEL
LIN {X 0,Y 530.891,Z 470.667,A -85,B 0,C 180,E1 -4221.435,E2 -4221.435} C_VEL
LIN {X 0,Y 530.69,Z 478.359,A -85,B 0,C 180,E1 -4222.581,E2 -4222.581} C_VEL
LIN {X 0,Y 530.606,Z 485.465,A -85,B 0,C 180,E1 -4223.917,E2 -4223.917} C_VEL
LIN {X 0,Y 530.459,Z 490.204,A -85,B 0,C 180,E1 -4225.06,E2 -4225.06} C_VEL
LIN {X 0,Y 530.516,Z 493.834,A -85,B 0,C 180,E1 -4226.202,E2 -4226.202} C_VEL
LIN {X 0,Y 530.457,Z 495.711,A -85,B 0,C 180,E1 -4226.962,E2 -4226.962} C_VEL
LIN {X 0,Y 530.411,Z 497.129,A -85,B 0,C 180,E1 -4227.722,E2 -4227.722} C_VEL
LIN {X 0,Y 530.344,Z 498.757,A -85,B 0,C 180,E1 -4229.241,E2 -4229.241} C_VEL
LIN {X 0,Y 530.343,Z 498.997,A -85,B 0,C 180,E1 -4230,E2 -4230} C_VEL
LIN {X 0,Y 530.344,Z 498.814,A -85,B 0,C 180,E1 -4230.759,E2 -4230.759} C_VEL
LIN {X 0,Y 530.412,Z 497.259,A -85,B 0,C 180,E1 -4232.278,E2 -4232.278} C_VEL
LIN {X 0,Y 530.457,Z 495.898,A -85,B 0,C 180,E1 -4233.038,E2 -4233.038} C_VEL
LIN {X 0,Y 530.523,Z 493.02,A -85,B 0,C 180,E1 -4234.178,E2 -4234.178} C_VEL
LIN {X 0,Y 530.524,Z 489.117,A -85,B 0,C 180,E1 -4235.321,E2 -4235.321} C_VEL
LIN {X 0,Y 530.593,Z 483.532,A -85,B 0,C 180,E1 -4236.576,E2 -4236.576} C_VEL
LIN {X 0,Y 530.758,Z 476.523,A -85,B 0,C 180,E1 -4237.801,E2 -4237.801} C_VEL
LIN {X 0,Y 530.903,Z 468.417,A -85,B 0,C 180,E1 -4238.949,E2 -4238.949} C_VEL
LIN {X 0,Y 531.117,Z 460.117,A -85,B 0,C 180,E1 -4239.906,E2 -4239.906} C_VEL
LIN {X 0,Y 531.404,Z 449.862,A -85,B 0,C 180,E1 -4240.863,E2 -4240.863} C_VEL
LIN {X 0,Y 531.678,Z 439.378,A -85,B 0,C 180,E1 -4241.651,E2 -4241.651} C_VEL
LIN {X 0,Y 531.883,Z 428.575,A -85,B 0,C 180,E1 -4242.302,E2 -4242.302} C_VEL
LIN {X 0,Y 532.113,Z 416.079,A -85,B 0,C 180,E1 -4242.878,E2 -4242.878} C_VEL
LIN {X 0,Y 532.048,Z 404.95,A -85,B 0,C 180,E1 -4243.256,E2 -4243.256} C_VEL
LIN {X 0,Y 530.46,Z 396.21,A -85,B 0,C 180,E1 -4243.528,E2 -4243.528} C_VEL
LIN {X 0,Y 530.478,Z 393.236,A -85,B 0,C 180,E1 -4246.154,E2 -4246.154} C_VEL
LIN {X 0,Y 530.469,Z 390.563,A -85,B 0,C 180,E1 -4248.54,E2 -4248.54} C_VEL
LIN {X 0,Y 530.501,Z 387.822,A -85,B 0,C 180,E1 -4250.959,E2 -4250.959} C_VEL
LIN {X 0,Y 530.566,Z 384.18,A -85,B 0,C 180,E1 -4254.245,E2 -4254.245} C_VEL
LIN {X 0,Y 530.619,Z 381.484,A -85,B 0,C 180,E1 -4256.765,E2 -4256.765} C_VEL
LIN {X 0,Y 530.666,Z 378.797,A -85,B 0,C 180,E1 -4259.342,E2 -4259.342} C_VEL
LIN {X 0,Y 530.715,Z 375.986,A -85,B 0,C 180,E1 -4262.057,E2 -4262.057} C_VEL
LIN {X 0,Y 530.728,Z 374.379,A -85,B 0,C 180,E1 -4263.792,E2 -4263.792} C_VEL
LIN {X 0,Y 530.916,Z 374.35,A -85,B 0,C 180,E1 -4266.148,E2 -4266.148} C_VEL
LIN {X 0,Y 530.971,Z 374.348,A -85,B 0,C 180,E1 -4268.654,E2 -4268.654} C_VEL
LIN {X 0,Y 531.001,Z 374.338,A -85,B 0,C 180,E1 -4271.435,E2 -4271.435} C_VEL
LIN {X 0,Y 530.981,Z 374.343,A -85,B 0,C 180,E1 -4274.548,E2 -4274.548} C_VEL
LIN {X 0,Y 530.986,Z 374.343,A -85,B 0,C 180,E1 -4277.834,E2 -4277.834} C_VEL
LIN {X 0,Y 530.994,Z 374.344,A -85,B 0,C 180,E1 -4280.557,E2 -4280.557} C_VEL
LIN {X 0,Y 530.97,Z 374.342,A -85,B 0,C 180,E1 -4283.442,E2 -4283.442} C_VEL
LIN {X 0,Y 531.005,Z 374.34,A -85,B 0,C 180,E1 -4286.494,E2 -4286.494} C_VEL
LIN {X 0,Y 530.979,Z 374.346,A -85,B 0,C 180,E1 -4289.355,E2 -4289.355} C_VEL
LIN {X 0,Y 531.018,Z 374.341,A -85,B 0,C 180,E1 -4292.468,E2 -4292.468} C_VEL
LIN {X 0,Y 531,Z 374.34,A -85,B 0,C 180,E1 -4294.942,E2 -4294.942} C_VEL
LIN {X 0,Y 530.977,Z 374.344,A -85,B 0,C 180,E1 -4298.247,E2 -4298.247} C_VEL
LIN {X 0,Y 531,Z 374.34,A -85,B 0,C 180,E1 -4300.677,E2 -4300.677} C_VEL
LIN {X 0,Y 530.979,Z 374.346,A -85,B 0,C 180,E1 -4303.071,E2 -4303.071} C_VEL
LIN {X 0,Y 531.025,Z 374.337,A -85,B 0,C 180,E1 -4305.436,E2 -4305.436} C_VEL
LIN {X 0,Y 531.043,Z 374.335,A -85,B 0,C 180,E1 -4308.55,E2 -4308.55} C_VEL
LIN {X 0,Y 531.042,Z 374.34,A -85,B 0,C 180,E1 -4311.629,E2 -4311.629} C_VEL
LIN {X 0,Y 531.126,Z 374.327,A -85,B 0,C 180,E1 -4314.685,E2 -4314.685} C_VEL
LIN {X 0,Y 531.141,Z 374.323,A -85,B 0,C 180,E1 -4317.725,E2 -4317.725} C_VEL
LIN {X 0,Y 531.158,Z 374.32,A -85,B 0,C 180,E1 -4320.758,E2 -4320.758} C_VEL
LIN {X 0,Y 531.109,Z 374.326,A -85,B 0,C 180,E1 -4323.034,E2 -4323.034} C_VEL
LIN {X 0,Y 531.088,Z 374.328,A -85,B 0,C 180,E1 -4326.077,E2 -4326.077} C_VEL
LIN {X 0,Y 531.036,Z 374.337,A -85,B 0,C 180,E1 -4329.138,E2 -4329.138} C_VEL
LIN {X 0,Y 531.047,Z 374.337,A -85,B 0,C 180,E1 -4332.225,E2 -4332.225} C_VEL
LIN {X 0,Y 531,Z 374.343,A -85,B 0,C 180,E1 -4335.35,E2 -4335.35} C_VEL
LIN {X 0,Y 530.992,Z 374.342,A -85,B 0,C 180,E1 -4338.521,E2 -4338.521} C_VEL
LIN {X 0,Y 531.006,Z 374.342,A -85,B 0,C 180,E1 -4340.938,E2 -4340.938} C_VEL
LIN {X 0,Y 530.97,Z 374.347,A -85,B 0,C 180,E1 -4344.225,E2 -4344.225} C_VEL
LIN {X 0,Y 531.01,Z 374.338,A -85,B 0,C 180,E1 -4346.743,E2 -4346.743} C_VEL
LIN {X 0,Y 530.987,Z 374.345,A -85,B 0,C 180,E1 -4349.322,E2 -4349.322} C_VEL
LIN {X 0,Y 530.97,Z 374.344,A -85,B 0,C 180,E1 -4352.1,E2 -4352.1} C_VEL
LIN {X 0,Y 530.975,Z 374.344,A -85,B 0,C 180,E1 -4354.851,E2 -4354.851} C_VEL
LIN {X 0,Y 530.97,Z 374.348,A -85,B 0,C 180,E1 -4357.507,E2 -4357.507} C_VEL
LIN {X 0,Y 530.986,Z 374.341,A -85,B 0,C 180,E1 -4360.433,E2 -4360.433} C_VEL
LIN {X 0,Y 530.969,Z 374.345,A -85,B 0,C 180,E1 -4363.494,E2 -4363.494} C_VEL
LIN {X 0,Y 530.971,Z 374.348,A -85,B 0,C 180,E1 -4366.506,E2 -4366.506} C_VEL
LIN {X 0,Y 530.99,Z 374.342,A -85,B 0,C 180,E1 -4368.976,E2 -4368.976} C_VEL
LIN {X 0,Y 530.993,Z 374.45,A -85,B 0,C 180,E1 -4371.894,E2 -4371.894} C_VEL
LIN {X 0,Y 531.999,Z 380.459,A -85,B 0,C 180,E1 -4374.091,E2 -4374.091} C_VEL
LIN {X 0,Y 531.987,Z 386.985,A -85,B 0,C 180,E1 -4376.334,E2 -4376.334} C_VEL
LIN {X 0,Y 531.76,Z 395.762,A -85,B 0,C 180,E1 -4379.213,E2 -4379.213} C_VEL
LIN {X 0,Y 531.544,Z 405.689,A -85,B 0,C 180,E1 -4382.434,E2 -4382.434} C_VEL
LIN {X 0,Y 531.313,Z 416.281,A -85,B 0,C 180,E1 -4385.791,E2 -4385.791} C_VEL
LIN {X 0,Y 531.094,Z 425.548,A -85,B 0,C 180,E1 -4388.659,E2 -4388.659} C_VEL
LIN {X 0,Y 530.959,Z 434.815,A -85,B 0,C 180,E1 -4391.477,E2 -4391.477} C_VEL
LIN {X 0,Y 530.787,Z 445.407,A -85,B 0,C 180,E1 -4394.644,E2 -4394.644} C_VEL
LIN {X 0,Y 530.722,Z 451.72,A -85,B 0,C 180,E1 -4396.472,E2 -4396.472} C_VEL
LIN {X 0,Y 532.303,Z 462.346,A -85,B 0,C 180,E1 -4396.738,E2 -4396.738} C_VEL
LIN {X 0,Y 532.153,Z 474.471,A -85,B 0,C 180,E1 -4397.123,E2 -4397.123} C_VEL
LIN {X 0,Y 531.936,Z 485.485,A -85,B 0,C 180,E1 -4397.602,E2 -4397.602} C_VEL
LIN {X 0,Y 531.701,Z 496.902,A -85,B 0,C 180,E1 -4398.247,E2 -4398.247} C_VEL
LIN {X 0,Y 531.465,Z 507.923,A -85,B 0,C 180,E1 -4399.042,E2 -4399.042} C_VEL
LIN {X 0,Y 531.195,Z 517.599,A -85,B 0,C 180,E1 -4399.903,E2 -4399.903} C_VEL
LIN {X 0,Y 530.969,Z 526.412,A -85,B 0,C 180,E1 -4400.861,E2 -4400.861} C_VEL
LIN {X 0,Y 530.779,Z 535.001,A -85,B 0,C 180,E1 -4402.008,E2 -4402.008} C_VEL
LIN {X 0,Y 530.637,Z 541.867,A -85,B 0,C 180,E1 -4403.154,E2 -4403.154} C_VEL
LIN {X 0,Y 530.611,Z 547.365,A -85,B 0,C 180,E1 -4404.299,E2 -4404.299} C_VEL
LIN {X 0,Y 530.457,Z 551.677,A -85,B 0,C 180,E1 -4405.44,E2 -4405.44} C_VEL
LIN {X 0,Y 530.516,Z 553.957,A -85,B 0,C 180,E1 -4406.202,E2 -4406.202} C_VEL
LIN {X 0,Y 530.457,Z 555.808,A -85,B 0,C 180,E1 -4406.962,E2 -4406.962} C_VEL
LIN {X 0,Y 530.411,Z 557.197,A -85,B 0,C 180,E1 -4407.722,E2 -4407.722} C_VEL
LIN {X 0,Y 530.344,Z 558.785,A -85,B 0,C 180,E1 -4409.241,E2 -4409.241} C_VEL
LIN {X 0,Y 530.342,Z 559,A -85,B 0,C 180,E1 -4410,E2 -4410} C_VEL
LIN {X 0,Y 530.361,Z 558.186,A -85,B 0,C 180,E1 -4411.519,E2 -4411.519} C_VEL
LIN {X 0,Y 530.411,Z 557.199,A -85,B 0,C 180,E1 -4412.278,E2 -4412.278} C_VEL
LIN {X 0,Y 530.457,Z 555.81,A -85,B 0,C 180,E1 -4413.038,E2 -4413.038} C_VEL
LIN {X 0,Y 530.522,Z 552.896,A -85,B 0,C 180,E1 -4414.178,E2 -4414.178} C_VEL
LIN {X 0,Y 530.524,Z 548.949,A -85,B 0,C 180,E1 -4415.321,E2 -4415.321} C_VEL
LIN {X 0,Y 530.599,Z 543.264,A -85,B 0,C 180,E1 -4416.582,E2 -4416.582} C_VEL
LIN {X 0,Y 530.758,Z 536.237,A -85,B 0,C 180,E1 -4417.801,E2 -4417.801} C_VEL
LIN {X 0,Y 530.931,Z 527.991,A -85,B 0,C 180,E1 -4418.948,E2 -4418.948} C_VEL
LIN {X 0,Y 531.119,Z 519.539,A -85,B 0,C 180,E1 -4419.905,E2 -4419.905} C_VEL
LIN {X 0,Y 531.421,Z 509.098,A -85,B 0,C 180,E1 -4420.863,E2 -4420.863} C_VEL
LIN {X 0,Y 531.69,Z 498.377,A -85,B 0,C 180,E1 -4421.655,E2 -4421.655} C_VEL
LIN {X 0,Y 531.89,Z 487.409,A -85,B 0,C 180,E1 -4422.302,E2 -4422.302} C_VEL
LIN {X 0,Y 532.133,Z 475.763,A -85,B 0,C 180,E1 -4422.829,E2 -4422.829} C_VEL
LIN {X 0,Y 532.303,Z 462.347,A -85,B 0,C 180,E1 -4423.262,E2 -4423.262} C_VEL
LIN {X 0,Y 530.71,Z 451.53,A -85,B 0,C 180,E1 -4423.546,E2 -4423.546} C_VEL
LIN {X 0,Y 530.818,Z 442.759,A -85,B 0,C 180,E1 -4426.143,E2 -4426.143} C_VEL
LIN {X 0,Y 530.959,Z 433.492,A -85,B 0,C 180,E1 -4428.923,E2 -4428.923} C_VEL
LIN {X 0,Y 531.118,Z 424.225,A -85,B 0,C 180,E1 -4431.747,E2 -4431.747} C_VEL
LIN {X 0,Y 531.343,Z 414.957,A -85,B 0,C 180,E1 -4434.623,E2 -4434.623} C_VEL
LIN {X 0,Y 531.539,Z 405.46,A -85,B 0,C 180,E1 -4437.64,E2 -4437.64} C_VEL
LIN {X 0,Y 531.791,Z 395.021,A -85,B 0,C 180,E1 -4441.025,E2 -4441.025} C_VEL
LIN {X 0,Y 531.987,Z 386.865,A -85,B 0,C 180,E1 -4443.701,E2 -4443.701} C_VEL
LIN {X 0,Y 532.002,Z 380.414,A -85,B 0,C 180,E1 -4445.91,E2 -4445.91} C_VEL
LIN {X 0,Y 530.985,Z 374.347,A -85,B 0,C 180,E1 -4448.166,E2 -4448.166} C_VEL
LIN {X 0,Y 530.989,Z 374.343,A -85,B 0,C 180,E1 -4451.024,E2 -4451.024} C_VEL
LIN {X 0,Y 530.97,Z 374.35,A -85,B 0,C 180,E1 -4453.494,E2 -4453.494} C_VEL
LIN {X 0,Y 530.958,Z 374.345,A -85,B 0,C 180,E1 -4456.504,E2 -4456.504} C_VEL
LIN {X 0,Y 530.99,Z 374.345,A -85,B 0,C 180,E1 -4458.976,E2 -4458.976} C_VEL
LIN {X 0,Y 530.962,Z 374.344,A -85,B 0,C 180,E1 -4461.53,E2 -4461.53} C_VEL
LIN {X 0,Y 530.979,Z 374.345,A -85,B 0,C 180,E1 -4464.382,E2 -4464.382} C_VEL
LIN {X 0,Y 530.97,Z 374.347,A -85,B 0,C 180,E1 -4467.134,E2 -4467.134} C_VEL
LIN {X 0,Y 530.973,Z 374.342,A -85,B 0,C 180,E1 -4469.803,E2 -4469.803} C_VEL
LIN {X 0,Y 531.019,Z 374.341,A -85,B 0,C 180,E1 -4472.467,E2 -4472.467} C_VEL
LIN {X 0,Y 530.999,Z 374.34,A -85,B 0,C 180,E1 -4474.942,E2 -4474.942} C_VEL
LIN {X 0,Y 530.976,Z 374.344,A -85,B 0,C 180,E1 -4478.247,E2 -4478.247} C_VEL
LIN {X 0,Y 531,Z 374.342,A -85,B 0,C 180,E1 -4480.677,E2 -4480.677} C_VEL
LIN {X 0,Y 530.99,Z 374.343,A -85,B 0,C 180,E1 -4483.071,E2 -4483.071} C_VEL
LIN {X 0,Y 531.024,Z 374.336,A -85,B 0,C 180,E1 -4485.436,E2 -4485.436} C_VEL
LIN {X 0,Y 531.053,Z 374.334,A -85,B 0,C 180,E1 -4488.55,E2 -4488.55} C_VEL
LIN {X 0,Y 531.061,Z 374.336,A -85,B 0,C 180,E1 -4491.63,E2 -4491.63} C_VEL
LIN {X 0,Y 531.124,Z 374.33,A -85,B 0,C 180,E1 -4494.685,E2 -4494.685} C_VEL
LIN {X 0,Y 531.143,Z 374.321,A -85,B 0,C 180,E1 -4497.725,E2 -4497.725} C_VEL
LIN {X 0,Y 531.157,Z 374.32,A -85,B 0,C 180,E1 -4500.758,E2 -4500.758} C_VEL
LIN {X 0,Y 531.108,Z 374.329,A -85,B 0,C 180,E1 -4503.034,E2 -4503.034} C_VEL
LIN {X 0,Y 531.087,Z 374.329,A -85,B 0,C 180,E1 -4506.077,E2 -4506.077} C_VEL
LIN {X 0,Y 531.053,Z 374.338,A -85,B 0,C 180,E1 -4508.371,E2 -4508.371} C_VEL
LIN {X 0,Y 531.056,Z 374.335,A -85,B 0,C 180,E1 -4511.672,E2 -4511.672} C_VEL
LIN {X 0,Y 531.035,Z 374.338,A -85,B 0,C 180,E1 -4514.956,E2 -4514.956} C_VEL
LIN {X 0,Y 530.985,Z 374.342,A -85,B 0,C 180,E1 -4517.724,E2 -4517.724} C_VEL
LIN {X 0,Y 531.029,Z 374.339,A -85,B 0,C 180,E1 -4520.127,E2 -4520.127} C_VEL
LIN {X 0,Y 530.949,Z 374.346,A -85,B 0,C 180,E1 -4522.573,E2 -4522.573} C_VEL
LIN {X 0,Y 530.999,Z 374.34,A -85,B 0,C 180,E1 -4525.058,E2 -4525.058} C_VEL
LIN {X 0,Y 531.02,Z 374.341,A -85,B 0,C 180,E1 -4527.595,E2 -4527.595} C_VEL
LIN {X 0,Y 530.978,Z 374.347,A -85,B 0,C 180,E1 -4530.645,E2 -4530.645} C_VEL
LIN {X 0,Y 530.991,Z 374.343,A -85,B 0,C 180,E1 -4533.773,E2 -4533.773} C_VEL
LIN {X 0,Y 530.959,Z 374.344,A -85,B 0,C 180,E1 -4536.558,E2 -4536.558} C_VEL
LIN {X 0,Y 530.993,Z 374.346,A -85,B 0,C 180,E1 -4539.443,E2 -4539.443} C_VEL
LIN {X 0,Y 530.982,Z 374.346,A -85,B 0,C 180,E1 -4542.457,E2 -4542.457} C_VEL
LIN {X 0,Y 530.955,Z 374.345,A -85,B 0,C 180,E1 -4543.564,E2 -4543.564} C_VEL
LIN {X 0,Y 530.284,Z 374.433,A -85,B 0,C 180,E1 -4544.198,E2 -4544.198} C_VEL
LIN {X 0,Y 527.442,Z 374.783,A -85,B 0,C 180,E1 -4545.226,E2 -4545.226} C_VEL
LIN {X 0,Y 525.043,Z 375.087,A -85,B 0,C 180,E1 -4546.055,E2 -4546.055} C_VEL
LIN {X 0,Y 524.012,Z 375.211,A -85,B 0,C 180,E1 -4546.695,E2 -4546.695} C_VEL
LIN {X 0,Y 523.926,Z 375.22,A -85,B 0,C 180,E1 -4546.911,E2 -4546.911} C_VEL
LIN {X 0,Y 523.952,Z 375.219,A -85,B 0,C 180,E1 -4549.921,E2 -4549.921} C_VEL
LIN {X 0,Y 523.906,Z 375.226,A -85,B 0,C 180,E1 -4552.867,E2 -4552.867} C_VEL
LIN {X 0,Y 523.763,Z 375.247,A -85,B 0,C 180,E1 -4555.697,E2 -4555.697} C_VEL
LIN {X 0,Y 523.674,Z 375.258,A -85,B 0,C 180,E1 -4556.616,E2 -4556.616} C_VEL
LIN {X 0,Y 523.633,Z 377.997,A -85,B 0,C 180,E1 -4559.335,E2 -4559.335} C_VEL
LIN {X 0,Y 523.608,Z 381.128,A -85,B 0,C 180,E1 -4562.359,E2 -4562.359} C_VEL
LIN {X 0,Y 523.521,Z 384.346,A -85,B 0,C 180,E1 -4565.408,E2 -4565.408} C_VEL
LIN {X 0,Y 523.461,Z 387.057,A -85,B 0,C 180,E1 -4567.918,E2 -4567.918} C_VEL
LIN {X 0,Y 523.433,Z 389.803,A -85,B 0,C 180,E1 -4570.387,E2 -4570.387} C_VEL
LIN {X 0,Y 523.409,Z 392.539,A -85,B 0,C 180,E1 -4572.818,E2 -4572.818} C_VEL
LIN {X 0,Y 523.382,Z 396.227,A -85,B 0,C 180,E1 -4576.013,E2 -4576.013} C_VEL
LIN {X 0,Y 523.403,Z 396.738,A -85,B 0,C 180,E1 -4576.397,E2 -4576.397} C_VEL
LIN {X 0,Y 525.377,Z 407.676,A -85,B 0,C 180,E1 -4576.732,E2 -4576.732} C_VEL
LIN {X 0,Y 525.116,Z 421.272,A -85,B 0,C 180,E1 -4577.242,E2 -4577.242} C_VEL
LIN {X 0,Y 524.933,Z 431.887,A -85,B 0,C 180,E1 -4577.784,E2 -4577.784} C_VEL
LIN {X 0,Y 524.642,Z 443.015,A -85,B 0,C 180,E1 -4578.506,E2 -4578.506} C_VEL
LIN {X 0,Y 524.377,Z 453.673,A -85,B 0,C 180,E1 -4579.381,E2 -4579.381} C_VEL
LIN {X 0,Y 524.086,Z 463.259,A -85,B 0,C 180,E1 -4580.35,E2 -4580.35} C_VEL
LIN {X 0,Y 523.903,Z 471.102,A -85,B 0,C 180,E1 -4581.32,E2 -4581.32} C_VEL
LIN {X 0,Y 523.678,Z 478.773,A -85,B 0,C 180,E1 -4582.481,E2 -4582.481} C_VEL
LIN {X 0,Y 523.542,Z 485.798,A -85,B 0,C 180,E1 -4583.835,E2 -4583.835} C_VEL
LIN {X 0,Y 523.384,Z 490.484,A -85,B 0,C 180,E1 -4584.993,E2 -4584.993} C_VEL
LIN {X 0,Y 523.444,Z 494.061,A -85,B 0,C 180,E1 -4586.151,E2 -4586.151} C_VEL
LIN {X 0,Y 523.368,Z 495.917,A -85,B 0,C 180,E1 -4586.921,E2 -4586.921} C_VEL
LIN {X 0,Y 523.335,Z 497.316,A -85,B 0,C 180,E1 -4587.691,E2 -4587.691} C_VEL
LIN {X 0,Y 523.25,Z 498.926,A -85,B 0,C 180,E1 -4589.23,E2 -4589.23} C_VEL
LIN {X 0,Y 523.247,Z 499.163,A -85,B 0,C 180,E1 -4590,E2 -4590} C_VEL
LIN {X 0,Y 523.25,Z 498.981,A -85,B 0,C 180,E1 -4590.77,E2 -4590.77} C_VEL
LIN {X 0,Y 523.335,Z 497.443,A -85,B 0,C 180,E1 -4592.309,E2 -4592.309} C_VEL
LIN {X 0,Y 523.368,Z 496.098,A -85,B 0,C 180,E1 -4593.079,E2 -4593.079} C_VEL
LIN {X 0,Y 523.442,Z 493.255,A -85,B 0,C 180,E1 -4594.235,E2 -4594.235} C_VEL
LIN {X 0,Y 523.463,Z 489.403,A -85,B 0,C 180,E1 -4595.393,E2 -4595.393} C_VEL
LIN {X 0,Y 523.522,Z 484.306,A -85,B 0,C 180,E1 -4596.579,E2 -4596.579} C_VEL
LIN {X 0,Y 523.7,Z 478.163,A -85,B 0,C 180,E1 -4597.712,E2 -4597.712} C_VEL
LIN {X 0,Y 523.901,Z 470.313,A -85,B 0,C 180,E1 -4598.875,E2 -4598.875} C_VEL
LIN {X 0,Y 524.154,Z 460.542,A -85,B 0,C 180,E1 -4600.039,E2 -4600.039} C_VEL
LIN {X 0,Y 524.456,Z 450.286,A -85,B 0,C 180,E1 -4601.009,E2 -4601.009} C_VEL
LIN {X 0,Y 524.783,Z 439.142,A -85,B 0,C 180,E1 -4601.852,E2 -4601.852} C_VEL
LIN {X 0,Y 524.97,Z 428.995,A -85,B 0,C 180,E1 -4602.467,E2 -4602.467} C_VEL
LIN {X 0,Y 525.22,Z 416.494,A -85,B 0,C 180,E1 -4603.05,E2 -4603.05} C_VEL
LIN {X 0,Y 525.239,Z 406.357,A -85,B 0,C 180,E1 -4603.404,E2 -4603.404} C_VEL
LIN {X 0,Y 523.368,Z 396.604,A -85,B 0,C 180,E1 -4603.715,E2 -4603.715} C_VEL
LIN {X 0,Y 523.397,Z 393.571,A -85,B 0,C 180,E1 -4606.379,E2 -4606.379} C_VEL
LIN {X 0,Y 523.414,Z 390.84,A -85,B 0,C 180,E1 -4608.799,E2 -4608.799} C_VEL
LIN {X 0,Y 523.42,Z 388.076,A -85,B 0,C 180,E1 -4611.256,E2 -4611.256} C_VEL
LIN {X 0,Y 523.497,Z 384.946,A -85,B 0,C 180,E1 -4614.089,E2 -4614.089} C_VEL
LIN {X 0,Y 523.546,Z 382.613,A -85,B 0,C 180,E1 -4616.295,E2 -4616.295} C_VEL
LIN {X 0,Y 523.62,Z 379.919,A -85,B 0,C 180,E1 -4618.894,E2 -4618.894} C_VEL
LIN {X 0,Y 523.626,Z 377.17,A -85,B 0,C 180,E1 -4621.564,E2 -4621.564} C_VEL
LIN {X 0,Y 523.675,Z 375.314,A -85,B 0,C 180,E1 -4623.384,E2 -4623.384} C_VEL
LIN {X 0,Y 523.852,Z 375.234,A -85,B 0,C 180,E1 -4625.232,E2 -4625.232} C_VEL
LIN {X 0,Y 523.92,Z 375.222,A -85,B 0,C 180,E1 -4628.102,E2 -4628.102} C_VEL
LIN {X 0,Y 523.945,Z 375.218,A -85,B 0,C 180,E1 -4631.092,E2 -4631.092} C_VEL
LIN {X 0,Y 523.939,Z 375.223,A -85,B 0,C 180,E1 -4634.229,E2 -4634.229} C_VEL
LIN {X 0,Y 523.921,Z 375.223,A -85,B 0,C 180,E1 -4636.833,E2 -4636.833} C_VEL
LIN {X 0,Y 523.944,Z 375.223,A -85,B 0,C 180,E1 -4638.908,E2 -4638.908} C_VEL
LIN {X 0,Y 523.922,Z 375.222,A -85,B 0,C 180,E1 -4641.898,E2 -4641.898} C_VEL
LIN {X 0,Y 523.94,Z 375.218,A -85,B 0,C 180,E1 -4644.91,E2 -4644.91} C_VEL
LIN {X 0,Y 523.94,Z 375.224,A -85,B 0,C 180,E1 -4647.68,E2 -4647.68} C_VEL
LIN {X 0,Y 523.959,Z 375.22,A -85,B 0,C 180,E1 -4650.677,E2 -4650.677} C_VEL
LIN {X 0,Y 523.979,Z 375.214,A -85,B 0,C 180,E1 -4653.729,E2 -4653.729} C_VEL
LIN {X 0,Y 523.918,Z 375.226,A -85,B 0,C 180,E1 -4656.27,E2 -4656.27} C_VEL
LIN {X 0,Y 523.952,Z 375.217,A -85,B 0,C 180,E1 -4658.767,E2 -4658.767} C_VEL
LIN {X 0,Y 523.955,Z 375.22,A -85,B 0,C 180,E1 -4661.221,E2 -4661.221} C_VEL
LIN {X 0,Y 523.936,Z 375.221,A -85,B 0,C 180,E1 -4663.639,E2 -4663.639} C_VEL
LIN {X 0,Y 523.945,Z 375.221,A -85,B 0,C 180,E1 -4666.028,E2 -4666.028} C_VEL
LIN {X 0,Y 524.018,Z 375.211,A -85,B 0,C 180,E1 -4668.394,E2 -4668.394} C_VEL
LIN {X 0,Y 523.994,Z 375.217,A -85,B 0,C 180,E1 -4671.516,E2 -4671.516} C_VEL
LIN {X 0,Y 524.051,Z 375.206,A -85,B 0,C 180,E1 -4673.841,E2 -4673.841} C_VEL
LIN {X 0,Y 524.075,Z 375.206,A -85,B 0,C 180,E1 -4676.925,E2 -4676.925} C_VEL
LIN {X 0,Y 524.119,Z 375.202,A -85,B 0,C 180,E1 -4680,E2 -4680} C_VEL
LIN {X 0,Y 524.075,Z 375.202,A -85,B 0,C 180,E1 -4683.075,E2 -4683.075} C_VEL
LIN {X 0,Y 524.051,Z 375.205,A -85,B 0,C 180,E1 -4686.159,E2 -4686.159} C_VEL
LIN {X 0,Y 524.004,Z 375.212,A -85,B 0,C 180,E1 -4689.262,E2 -4689.262} C_VEL
LIN {X 0,Y 524.031,Z 375.211,A -85,B 0,C 180,E1 -4691.751,E2 -4691.751} C_VEL
LIN {X 0,Y 523.999,Z 375.212,A -85,B 0,C 180,E1 -4695.052,E2 -4695.052} C_VEL
LIN {X 0,Y 523.953,Z 375.217,A -85,B 0,C 180,E1 -4697.969,E2 -4697.969} C_VEL
LIN {X 0,Y 523.978,Z 375.217,A -85,B 0,C 180,E1 -4700.41,E2 -4700.41} C_VEL
LIN {X 0,Y 523.915,Z 375.224,A -85,B 0,C 180,E1 -4702.893,E2 -4702.893} C_VEL
LIN {X 0,Y 523.989,Z 375.215,A -85,B 0,C 180,E1 -4706.02,E2 -4706.02} C_VEL
LIN {X 0,Y 523.944,Z 375.22,A -85,B 0,C 180,E1 -4708.874,E2 -4708.874} C_VEL
LIN {X 0,Y 523.926,Z 375.221,A -85,B 0,C 180,E1 -4711.544,E2 -4711.544} C_VEL
LIN {X 0,Y 523.938,Z 375.223,A -85,B 0,C 180,E1 -4714.29,E2 -4714.29} C_VEL
LIN {X 0,Y 523.911,Z 375.224,A -85,B 0,C 180,E1 -4717.132,E2 -4717.132} C_VEL
LIN {X 0,Y 523.941,Z 375.218,A -85,B 0,C 180,E1 -4720.13,E2 -4720.13} C_VEL
LIN {X 0,Y 523.926,Z 375.225,A -85,B 0,C 180,E1 -4723.167,E2 -4723.167} C_VEL
LIN {X 0,Y 523.946,Z 375.219,A -85,B 0,C 180,E1 -4725.772,E2 -4725.772} C_VEL
LIN {X 0,Y 523.945,Z 375.22,A -85,B 0,C 180,E1 -4728.908,E2 -4728.908} C_VEL
LIN {X 0,Y 523.936,Z 375.315,A -85,B 0,C 180,E1 -4731.655,E2 -4731.655} C_VEL
LIN {X 0,Y 524.985,Z 381.362,A -85,B 0,C 180,E1 -4733.911,E2 -4733.911} C_VEL
LIN {X 0,Y 525.031,Z 387.572,A -85,B 0,C 180,E1 -4736.091,E2 -4736.091} C_VEL
LIN {X 0,Y 524.777,Z 396.324,A -85,B 0,C 180,E1 -4738.994,E2 -4738.994} C_VEL
LIN {X 0,Y 524.562,Z 406.072,A -85,B 0,C 180,E1 -4742.161,E2 -4742.161} C_VEL
LIN {X 0,Y 524.339,Z 414.957,A -85,B 0,C 180,E1 -4745.025,E2 -4745.025} C_VEL
LIN {X 0,Y 524.126,Z 424.224,A -85,B 0,C 180,E1 -4747.948,E2 -4747.948} C_VEL
LIN {X 0,Y 523.926,Z 433.491,A -85,B 0,C 180,E1 -4750.813,E2 -4750.813} C_VEL
LIN {X 0,Y 523.765,Z 442.759,A -85,B 0,C 180,E1 -4753.633,E2 -4753.633} C_VEL
LIN {X 0,Y 523.656,Z 451.72,A -85,B 0,C 180,E1 -4756.286,E2 -4756.286} C_VEL
LIN {X 0,Y 525.388,Z 462.346,A -85,B 0,C 180,E1 -4756.56,E2 -4756.56} C_VEL
LIN {X 0,Y 525.219,Z 475.766,A -85,B 0,C 180,E1 -4756.999,E2 -4756.999} C_VEL
LIN {X 0,Y 524.964,Z 487.407,A -85,B 0,C 180,E1 -4757.533,E2 -4757.533} C_VEL
LIN {X 0,Y 524.707,Z 498.61,A -85,B 0,C 180,E1 -4758.204,E2 -4758.204} C_VEL
LIN {X 0,Y 524.405,Z 510.259,A -85,B 0,C 180,E1 -4759.088,E2 -4759.088} C_VEL
LIN {X 0,Y 524.096,Z 519.537,A -85,B 0,C 180,E1 -4759.96,E2 -4759.96} C_VEL
LIN {X 0,Y 523.896,Z 527.99,A -85,B 0,C 180,E1 -4760.931,E2 -4760.931} C_VEL
LIN {X 0,Y 523.688,Z 536.236,A -85,B 0,C 180,E1 -4762.093,E2 -4762.093} C_VEL
LIN {X 0,Y 523.575,Z 541.868,A -85,B 0,C 180,E1 -4763.061,E2 -4763.061} C_VEL
LIN {X 0,Y 523.544,Z 547.365,A -85,B 0,C 180,E1 -4764.222,E2 -4764.222} C_VEL
LIN {X 0,Y 523.361,Z 551.677,A -85,B 0,C 180,E1 -4765.378,E2 -4765.378} C_VEL
LIN {X 0,Y 523.443,Z 553.957,A -85,B 0,C 180,E1 -4766.151,E2 -4766.151} C_VEL
LIN {X 0,Y 523.367,Z 555.808,A -85,B 0,C 180,E1 -4766.921,E2 -4766.921} C_VEL
LIN {X 0,Y 523.335,Z 557.197,A -85,B 0,C 180,E1 -4767.691,E2 -4767.691} C_VEL
LIN {X 0,Y 523.25,Z 558.785,A -85,B 0,C 180,E1 -4769.23,E2 -4769.23} C_VEL
LIN {X 0,Y 523.246,Z 559,A -85,B 0,C 180,E1 -4770,E2 -4770} C_VEL
LIN {X 0,Y 523.275,Z 558.186,A -85,B 0,C 180,E1 -4771.539,E2 -4771.539} C_VEL
LIN {X 0,Y 523.335,Z 557.199,A -85,B 0,C 180,E1 -4772.309,E2 -4772.309} C_VEL
LIN {X 0,Y 523.367,Z 555.81,A -85,B 0,C 180,E1 -4773.079,E2 -4773.079} C_VEL
LIN {X 0,Y 523.441,Z 552.896,A -85,B 0,C 180,E1 -4774.235,E2 -4774.235} C_VEL
LIN {X 0,Y 523.464,Z 548.949,A -85,B 0,C 180,E1 -4775.393,E2 -4775.393} C_VEL
LIN {X 0,Y 523.523,Z 543.727,A -85,B 0,C 180,E1 -4776.581,E2 -4776.581} C_VEL
LIN {X 0,Y 523.665,Z 537.468,A -85,B 0,C 180,E1 -4777.713,E2 -4777.713} C_VEL
LIN {X 0,Y 523.857,Z 529.478,A -85,B 0,C 180,E1 -4778.875,E2 -4778.875} C_VEL
LIN {X 0,Y 524.06,Z 521.335,A -85,B 0,C 180,E1 -4779.845,E2 -4779.845} C_VEL
LIN {X 0,Y 524.362,Z 511.4,A -85,B 0,C 180,E1 -4780.815,E2 -4780.815} C_VEL
LIN {X 0,Y 524.679,Z 500.201,A -85,B 0,C 180,E1 -4781.687,E2 -4781.687} C_VEL
LIN {X 0,Y 524.91,Z 489.176,A -85,B 0,C 180,E1 -4782.37,E2 -4782.37} C_VEL
LIN {X 0,Y 525.163,Z 476.978,A -85,B 0,C 180,E1 -4782.953,E2 -4782.953} C_VEL
LIN {X 0,Y 525.384,Z 464.175,A -85,B 0,C 180,E1 -4783.391,E2 -4783.391} C_VEL
LIN {X 0,Y 524.786,Z 458.365,A -85,B 0,C 180,E1 -4783.554,E2 -4783.554} C_VEL
LIN {X 0,Y 523.646,Z 451.53,A -85,B 0,C 180,E1 -4783.732,E2 -4783.732} C_VEL
LIN {X 0,Y 523.765,Z 442.759,A -85,B 0,C 180,E1 -4786.367,E2 -4786.367} C_VEL
LIN {X 0,Y 523.926,Z 433.492,A -85,B 0,C 180,E1 -4789.187,E2 -4789.187} C_VEL
LIN {X 0,Y 524.126,Z 424.225,A -85,B 0,C 180,E1 -4792.052,E2 -4792.052} C_VEL
LIN {X 0,Y 524.343,Z 414.957,A -85,B 0,C 180,E1 -4794.974,E2 -4794.974} C_VEL
LIN {X 0,Y 524.58,Z 405.69,A -85,B 0,C 180,E1 -4797.964,E2 -4797.964} C_VEL
LIN {X 0,Y 524.799,Z 396.312,A -85,B 0,C 180,E1 -4801.01,E2 -4801.01} C_VEL
LIN {X 0,Y 525.026,Z 387.569,A -85,B 0,C 180,E1 -4803.908,E2 -4803.908} C_VEL
LIN {X 0,Y 524.992,Z 381.309,A -85,B 0,C 180,E1 -4806.088,E2 -4806.088} C_VEL
LIN {X 0,Y 523.926,Z 375.227,A -85,B 0,C 180,E1 -4808.407,E2 -4808.407} C_VEL
LIN {X 0,Y 523.962,Z 375.218,A -85,B 0,C 180,E1 -4811.311,E2 -4811.311} C_VEL
LIN {X 0,Y 523.959,Z 375.221,A -85,B 0,C 180,E1 -4814.691,E2 -4814.691} C_VEL
LIN {X 0,Y 523.956,Z 375.215,A -85,B 0,C 180,E1 -4817.881,E2 -4817.881} C_VEL
LIN {X 0,Y 523.926,Z 375.223,A -85,B 0,C 180,E1 -4820.916,E2 -4820.916} C_VEL
LIN {X 0,Y 523.927,Z 375.224,A -85,B 0,C 180,E1 -4823.827,E2 -4823.827} C_VEL
LIN {X 0,Y 523.945,Z 375.219,A -85,B 0,C 180,E1 -4826.636,E2 -4826.636} C_VEL
LIN {X 0,Y 523.959,Z 375.219,A -85,B 0,C 180,E1 -4829.356,E2 -4829.356} C_VEL
LIN {X 0,Y 523.982,Z 375.216,A -85,B 0,C 180,E1 -4832.281,E2 -4832.281} C_VEL
LIN {X 0,Y 523.951,Z 375.221,A -85,B 0,C 180,E1 -4834.581,E2 -4834.581} C_VEL
LIN {X 0,Y 523.923,Z 375.225,A -85,B 0,C 180,E1 -4837.757,E2 -4837.757} C_VEL
LIN {X 0,Y 523.98,Z 375.215,A -85,B 0,C 180,E1 -4840.408,E2 -4840.408} C_VEL
LIN {X 0,Y 523.971,Z 375.22,A -85,B 0,C 180,E1 -4842.837,E2 -4842.837} C_VEL
LIN {X 0,Y 523.982,Z 375.213,A -85,B 0,C 180,E1 -4845.236,E2 -4845.236} C_VEL
LIN {X 0,Y 524.019,Z 375.211,A -85,B 0,C 180,E1 -4848.394,E2 -4848.394} C_VEL
LIN {X 0,Y 524.009,Z 375.214,A -85,B 0,C 180,E1 -4851.516,E2 -4851.516} C_VEL
LIN {X 0,Y 524.086,Z 375.205,A -85,B 0,C 180,E1 -4854.614,E2 -4854.614} C_VEL
LIN {X 0,Y 524.116,Z 375.197,A -85,B 0,C 180,E1 -4857.695,E2 -4857.695} C_VEL
LIN {X 0,Y 524.127,Z 375.196,A -85,B 0,C 180,E1 -4860.768,E2 -4860.768} C_VEL
LIN {X 0,Y 524.074,Z 375.206,A -85,B 0,C 180,E1 -4863.075,E2 -4863.075} C_VEL
LIN {X 0,Y 524.05,Z 375.206,A -85,B 0,C 180,E1 -4866.159,E2 -4866.159} C_VEL
LIN {X 0,Y 524.001,Z 375.216,A -85,B 0,C 180,E1 -4868.484,E2 -4868.484} C_VEL
LIN {X 0,Y 524.007,Z 375.213,A -85,B 0,C 180,E1 -4871.739,E2 -4871.739} C_VEL
LIN {X 0,Y 523.998,Z 375.215,A -85,B 0,C 180,E1 -4875.052,E2 -4875.052} C_VEL
LIN {X 0,Y 523.952,Z 375.218,A -85,B 0,C 180,E1 -4877.97,E2 -4877.97} C_VEL
LIN {X 0,Y 523.977,Z 375.22,A -85,B 0,C 180,E1 -4880.41,E2 -4880.41} C_VEL
LIN {X 0,Y 523.915,Z 375.221,A -85,B 0,C 180,E1 -4882.894,E2 -4882.894} C_VEL
LIN {X 0,Y 523.988,Z 375.215,A -85,B 0,C 180,E1 -4886.02,E2 -4886.02} C_VEL
LIN {X 0,Y 523.943,Z 375.222,A -85,B 0,C 180,E1 -4888.875,E2 -4888.875} C_VEL
LIN {X 0,Y 523.925,Z 375.221,A -85,B 0,C 180,E1 -4891.544,E2 -4891.544} C_VEL
LIN {X 0,Y 523.937,Z 375.223,A -85,B 0,C 180,E1 -4894.29,E2 -4894.29} C_VEL
LIN {X 0,Y 523.911,Z 375.223,A -85,B 0,C 180,E1 -4897.132,E2 -4897.132} C_VEL
LIN {X 0,Y 523.941,Z 375.219,A -85,B 0,C 180,E1 -4900.13,E2 -4900.13} C_VEL
LIN {X 0,Y 523.939,Z 375.223,A -85,B 0,C 180,E1 -4902.459,E2 -4902.459} C_VEL
LIN {X 0,Y 523.949,Z 375.218,A -85,B 0,C 180,E1 -4905.31,E2 -4905.31} C_VEL
LIN {X 0,Y 523.926,Z 375.22,A -85,B 0,C 180,E1 -4906.911,E2 -4906.911} C_VEL
LIN {X 0,Y 523.259,Z 375.308,A -85,B 0,C 180,E1 -4907.553,E2 -4907.553} C_VEL
LIN {X 0,Y 520.415,Z 375.659,A -85,B 0,C 180,E1 -4908.594,E2 -4908.594} C_VEL
LIN {X 0,Y 518.009,Z 375.962,A -85,B 0,C 180,E1 -4909.433,E2 -4909.433} C_VEL
LIN {X 0,Y 516.972,Z 376.087,A -85,B 0,C 180,E1 -4910.081,E2 -4910.081} C_VEL
LIN {X 0,Y 516.884,Z 376.097,A -85,B 0,C 180,E1 -4910.3,E2 -4910.3} C_VEL
LIN {X 0,Y 516.849,Z 376.105,A -85,B 0,C 180,E1 -4913.348,E2 -4913.348} C_VEL
